	GVL.Pro4_.Signal_In.T_Ts_Result_Scanner( IN:= GVL.X[31], PT := T#0MS);
	GVL.Pro4_.Signal_In.T_Ts_Pass( IN:= GVL.X[21], PT := T#10MS);
	GVL.Pro4_.Signal_In.T_Ts_Fail( IN:= GVL.X[22], PT := T#10MS);
	GVL.Pro4_.Signal_In.T_Door_ss( IN:= GVL.X[23], PT := T#100MS);
	GVL.Pro4_.Signal_In.T_Ts_Press_Up( IN:= GVL.X[24], PT := T#10MS);
	GVL.Pro4_.Signal_In.T_Ts_Check_Gap( IN:= GVL.X[25], PT := T#500MS);
	// CHECK TS 
	T_RESET_TS(IN := GVL.Pro4_.Man.D_Ts = 2 OR GVL.Pro4_.Man.D_Ts = 3,  PT := T#5S, Q =>);
	T_OUT_RESET_TS( IN := (GVL.Y[20] AND NOT GVL.Pro4_.Signal_In.T_Ts_Fail.Q AND NOT  GVL.Pro4_.Signal_In.T_Ts_Pass.Q), PT := T#20S, Q =>);
	IF GVL.Y[20] AND GVL.Pro4_.Man.D_Ts = 0 AND NOT GVL.Pro4_.Signal_In.T_Ts_Fail.Q AND NOT GVL.Pro4_.Signal_In.T_Ts_Pass.Q  THEN
		GVL.Pro4_.Man.D_Ts := 1;
	END_IF;
	IF GVL.Pro4_.Man.D_Ts = 1 AND GVL.Pro4_.Signal_In.T_Ts_Pass.Q THEN
		GVL.Pro4_.Man.D_Ts := 2;
	ELSIF GVL.Pro4_.Man.D_Ts = 1 AND GVL.Pro4_.Signal_In.T_Ts_Fail.Q THEN
		GVL.Pro4_.Man.D_Ts := 3;
	END_IF
	IF T_RESET_TS.Q OR T_OUT_RESET_TS.Q THEN
		GVL.Pro4_.Man.TS_On_Off := 0;
		GVL.Pro4_.Man.D_Ts := 0 ;
		T_OUT_RESET_TS.IN := FALSE;
		T_RESET_TS.IN := FALSE;
	END_IF
	// check Víison
	GVL.Pro4_.Signal_In.T_Vs_detect( IN:= GVL.X[26], PT := T#100MS);
	GVL.Pro4_.Signal_In.T_Vs_Result_Scanner( IN:= GVL.X[30], PT := T#1MS);
	GVL.Pro4_.Signal_In.T_Vs_Pass( IN:= GVL.X[32] AND GVL.Pro4_.Signal_In.T_Vs_detect.Q, PT := T#1000MS);
	GVL.Pro4_.Signal_In.T_Vs_Fail( IN:= GVL.X[33] AND GVL.Pro4_.Signal_In.T_Vs_detect.Q, PT := T#1000MS);
	// CHECK VS 
	T_RESET_VS(IN := GVL.Pro4_.Man.D_Vs = 2 OR GVL.Pro4_.Man.D_Vs = 3,  PT := T#5S, Q =>);
	T_OUT_RESET_VS( IN := GVL.Y[21] AND NOT GVL.Pro4_.Signal_In.T_Vs_Fail.Q AND NOT  GVL.Pro4_.Signal_In.T_Vs_Pass.Q, PT := T#20S, Q =>);
	IF GVL.Y[21] AND GVL.Pro4_.Man.D_Vs = 0 AND NOT GVL.Pro4_.Signal_In.T_Vs_Fail.Q AND NOT GVL.Pro4_.Signal_In.T_Vs_Pass.Q  THEN
		GVL.Pro4_.Man.D_Vs := 1;
	END_IF;
	IF GVL.Pro4_.Man.D_Vs = 1 AND GVL.Pro4_.Signal_In.T_Ts_Pass.Q THEN
		GVL.Pro4_.Man.D_Vs := 2;
	ELSIF GVL.Pro4_.Man.D_Vs = 1 AND GVL.Pro4_.Signal_In.T_Ts_Fail.Q THEN
		GVL.Pro4_.Man.D_Vs := 3;
	END_IF
	IF T_RESET_VS.Q AND T_OUT_RESET_VS.Q THEN
		GVL.Pro4_.Man.Vs_On_Off := 0;
		GVL.Pro4_.Man.D_Vs := 0 ;
		T_OUT_RESET_VS.IN := FALSE;
		T_RESET_VS.IN := FALSE;
	END_IF
	// Conveyor
	GVL.Pro4_.Signal_In.T_Cv_In_1( IN:= NOT GVL.X[27], PT := T#1500MS);
	GVL.Pro4_.Signal_In.T_Cv_In_2( IN:= not GVL.X[28], PT := T#500MS);
	GVL.Pro4_.Signal_In.T_Cv_OK_out( IN:= GVL.X[29], PT := T#500MS);
	
	GVL.Pro4_.Signal_In.T_Cv_NG_out_1( IN:= NOT GVL.X[40], PT := T#10MS);
	GVL.Pro4_.Signal_In.T_Cv_NG_out_2( IN:= NOT GVL.X[41], PT := T#10MS);
	GVL.Pro4_.Signal_In.T_Cv_NG_out_full( IN:= NOT GVL.X[42], PT := T#10MS);

END_IF;


//


RETURN;
END_ACTION

ACTION ACT_Manual_MC:

END_ACTION

ACTION ACT_Out:
// Share all robot
// green
GVL.Y[2] := GVL.HMI_MAIN.yStart AND NOT GVL.HMI_MAIN.yStop AND NOT GVL.HMI_MAIN.yLamp_Yellow AND NOT POU_MOTION.HeavyAlarm ;
// red
GVL.Y[0] := GVL.HMI_MAIN.yStop AND NOT GVL.HMI_MAIN.yStart OR POU_MOTION.HeavyAlarm;
// yellow
GVL.Y[1] := GVL.HMI_MAIN.yLamp_Yellow OR POU_MOTION.LightAlarm;
// buzz
GVL.Y[3] := GVL.HMI_MAIN.yBuzz;

// Tool 1 A
GVL.Y[4] := GVL.RB_A_.Tool_1 OR GVL.Y[4];
// Tool 2 A
GVL.Y[5] := GVL.RB_A_.Tool_2;
// Tool 1 B			
GVL.Y[6] := GVL.RB_B_.Tool_1;
// Tool 2 B
GVL.Y[7] := GVL.RB_B_.Tool_2;

// Project 3
IF GVL.ProjectAndModel.Project_No_Current = 3 THEN
	
	// PRoject 4
	IF GVL.RB_A.Auto OR GVL.RB_B.Auto THEN
		GVL.Pro4_.Man.TS_On_Off := 0;
		GVL.Pro4_.Man.Vs_On_Off := 0;
		GVL.Pro4_.Man.Trigger_Barcode_Ts_On_Off := 0;
		GVL.Pro4_.Man.Trigger_Barcode_Ts_On_Off := 0;
		GVL.Pro4_.Man.Cv_NG_On_Off := 0;
		GVL.Pro4_.Man.Lighting_On_Off := 0;
		GVL.Pro4_.Man.centering_ts_On_Off := 0;
	END_IF
	
	IF GVL.RB_A.Manual OR GVL.RB_B.Manual THEN
		GVL.Pro4_.Auto.TS_On_Off := 0;
		GVL.Pro4_.Auto.Vs_On_Off := 0;
		GVL.Pro4_.Auto.Trigger_Barcode_Ts_On_Off := 0;
		GVL.Pro4_.Auto.Trigger_Barcode_Ts_On_Off := 0;
		GVL.Pro4_.Auto.Cv_NG_On_Off := 0;
		GVL.Pro4_.Auto.Lighting_On_Off := 0;
		GVL.Pro4_.Auto.centering_ts_On_Off := 0;
	END_IF
	
	// centering test sóng
	GVL.Y[10] :=  (GVL.RB_A.Auto AND GVL.RB_B.Auto AND GVL.Pro4_.Auto.centering_ts_On_Off )OR 
				( ( GVL.RB_A.Manual OR GVL.RB_B.Manual) AND GVL.Pro4_.Man.centering_ts_On_Off );
	
	// test sóng
	GVL.Y[20] :=  (GVL.RB_A.Auto AND GVL.RB_B.Auto AND GVL.Pro4_.Auto.TS_On_Off )OR 
				( ( GVL.RB_A.Manual OR GVL.RB_B.Manual) AND GVL.Pro4_.Man.TS_On_Off );
	// test vision			
	GVL.Y[21] :=  (GVL.RB_A.Auto AND GVL.RB_B.Auto AND GVL.Pro4_.Auto.Vs_On_Off )OR 
				( ( GVL.RB_A.Manual OR GVL.RB_B.Manual) AND GVL.Pro4_.Man.Vs_On_Off );
	// trigger Barcode	ts			
	GVL.Y[22] :=  (GVL.RB_A.Auto AND GVL.RB_B.Auto AND GVL.Pro4_.Auto.Trigger_Barcode_Ts_On_Off )OR 
				( ( GVL.RB_A.Manual OR GVL.RB_B.Manual) AND GVL.Pro4_.Man.Trigger_Barcode_Ts_On_Off );
	// trigger Barcode vs
	GVL.Y[23] :=  (GVL.RB_A.Auto AND GVL.RB_B.Auto AND GVL.Pro4_.Auto.Trigger_Barcode_Vs_On_Off )OR 
				( ( GVL.RB_A.Manual OR GVL.RB_B.Manual) AND GVL.Pro4_.Man.Trigger_Barcode_Vs_On_Off );
	// Conveyor NG
	GVL.Y[27] :=  (GVL.RB_A.Auto AND GVL.RB_B.Auto AND GVL.Pro4_.Auto.Cv_NG_On_Off )OR 
				( ( GVL.RB_A.Manual OR GVL.RB_B.Manual) AND GVL.Pro4_.Man.Cv_NG_On_Off );			
	// Lighting vision align
	GVL.Y[28] :=  (GVL.RB_A.Auto AND GVL.RB_B.Auto AND GVL.Pro4_.Auto.Lighting_On_Off )OR 
				( ( GVL.RB_A.Manual OR GVL.RB_B.Manual) AND GVL.Pro4_.Man.Lighting_On_Off );			
			
END_IF;
END_ACTION

ACTION ACT_SAVE_FILE:
// Duyet de kiem tra tin hieu luu va doc du lieu CAM
FOR i_cam := 0 TO 10 BY 1 DO
	GVL.RTrig_Save_Data_Cam[i_cam](CLK := GVL.Save_Data_Cam[i_cam]);
	GVL.RTrig_Load_Data_Cam[i_cam](CLK := GVL.Load_Data_Cam[i_cam]);
	// Luu du lieu CAM
	IF GVL.RTrig_Save_Data_Cam[i_cam].Q THEN
		filedata.Save(    
			pData := ADR(GVL.Data_Calib_RB),
			uiSize := SIZEOF(GVL.Data_Calib_RB),
			sFileName := CONCAT('Data_Cam_',INT_TO_STRING(i_cam)));
	END_IF
	// Doc lai du lieu CAM
	IF GVL.RTrig_Load_Data_Cam[i_cam].Q THEN
		filedata.Load(    
			pData := ADR(GVL.Data_Calib_RB),
			uiSize := SIZEOF(GVL.Data_Calib_RB),
			sFileName := CONCAT('Data_Cam_',INT_TO_STRING(i_cam)));
		GVL.Load_Data_Cam[i_cam] := FALSE;
	END_IF
END_FOR

// Save All Tool Config to File
r_Save_ToolConfig(CLK := GVL.g_stHMITool_Config_Save_All);
IF r_Save_ToolConfig.Q THEN
	
	filedata.Save(    
	pData := ADR(GVL.g_aToolConfigA),
    uiSize := SIZEOF(GVL.g_aToolConfigA),
    sFileName := 'Tool_Config_A.bin');	
	GVL.g_stHMITool_Config_Save_All := FALSE;
END_IF

// Read Tool Config From File
r_Read_ToolConfig(CLK := GVL.g_stHMITool_Config_Read_All);
IF r_Read_ToolConfig.Q OR Read_Config_First THEN
	
	filedata.Load(    
	pData := ADR(GVL.g_aToolConfigA),
    uiSize := SIZEOF(GVL.g_aToolConfigA),
    sFileName := 'Tool_Config_A.bin');	
	GVL.g_stHMITool_Config_Read_All := FALSE;
	GVL.g_stHMIToolEditorA.LoadCommand := TRUE; // cho doc du lieu tool hien tai
END_IF


// Save Conveyor Config
r_Save_ConveyorConfig(CLK:= GVL.g_stHMIConveyor_Config_Save);
IF r_Save_ConveyorConfig.Q THEN
	filedata.Save(    
	pData := ADR(GVL.g_aConveyorRuntime),
    uiSize := SIZEOF(GVL.g_aConveyorRuntime),
    sFileName := 'Conveyor_Config.bin');
	
END_IF

// Read Conveyor Config
r_Read_ConveyorConfig(CLK:= GVL.g_stHMIConveyor_Config_Read);
IF r_Read_ConveyorConfig.Q OR Read_Config_First THEN
	filedata.Load(    
	pData := ADR(GVL.g_aConveyorRuntime),
    uiSize := SIZEOF(GVL.g_aConveyorRuntime),
    sFileName := 'Conveyor_Config.bin');
	GVL.g_stHMIConveyor_Config_Read := FALSE;
END_IF

// Save Tracking Config
r_Save_TrackingConfig(CLK:= GVL.g_stHMITracking_Config_Save);
IF r_Save_TrackingConfig.Q THEN
	filedata.Save(    
	pData := ADR(GVL.g_stTrackingConfig_A),
    uiSize := SIZEOF(GVL.g_stTrackingConfig_A),
    sFileName := 'TrackingConfig_A.bin');
END_IF

// Read Tracking Config
r_Read_TrackingConfig(CLK:= GVL.g_stHMITracking_Config_Read);
IF r_Read_TrackingConfig.Q OR Read_Config_First THEN
	filedata.Load(    
	pData := ADR(GVL.g_stTrackingConfig_A),
    uiSize := SIZEOF(GVL.g_stTrackingConfig_A),
    sFileName := 'TrackingConfig_A.bin');
	GVL.g_stHMITracking_Config_Read := FALSE;
END_IF

// Save All Senssor Source Config to File
//r_Save_ToolConfig(CLK := GVL.g_stHMITool_Config_Save_All);
IF GVL.g_xHMISaveSensorSourceA_All THEN
	
	filedata.Save(    
	pData := ADR(GVL.g_aSensorSourceConfigA),
    uiSize := SIZEOF(GVL.g_aSensorSourceConfigA),
    sFileName := 'SensorSource_Config_A.bin');	
	GVL.g_xHMISaveSensorSourceA_All := FALSE;	
END_IF

// Read Tool Config From File
IF GVL.g_xHMILoadSensorSourceA_All OR Read_Config_First THEN
	
	filedata.Load(    
	pData := ADR(GVL.g_aSensorSourceConfigA),
    uiSize := SIZEOF(GVL.g_aSensorSourceConfigA),
    sFileName := 'SensorSource_Config_A.bin');	
	GVL.g_xHMILoadSensorSourceA_All := FALSE;
	GVL.g_xHMILoadSensorSourceA := TRUE; // cho doc du lieu senssor source hien tai
END_IF

// Save All Recipe Config to File
IF GVL.g_xHMISaveTrackingRecipeA_All THEN
	
	filedata.Save(    
	pData := ADR(GVL.g_aMultiTrackRecipeA),
    uiSize := SIZEOF(GVL.g_aMultiTrackRecipeA),
    sFileName := 'MultiTrackRecipe_Config_A.bin');	
	GVL.g_xHMISaveTrackingRecipeA_All := FALSE;	
END_IF

// Read Tool Config From File
IF GVL.g_xHMILoadTrackingRecipeA_All OR Read_Config_First THEN
	
	filedata.Load(    
	pData := ADR(GVL.g_aMultiTrackRecipeA),
    uiSize := SIZEOF(GVL.g_aMultiTrackRecipeA),
    sFileName := 'MultiTrackRecipe_Config_A.bin');	
	GVL.g_xHMILoadTrackingRecipeA_All := FALSE;
	GVL.g_xHMILoadTrackingRecipeA := TRUE; // cho doc du lieu senssor source hien tai
END_IF




//=============================================================================
// SAVE ALL VISION TRACKING SOURCE CONFIG
//=============================================================================
IF GVL.g_xHMISaveAllVisionSourceA THEN

    filedata.Save(
        pData := ADR(GVL.g_aVisionTrackingSourceConfigA),
        uiSize := SIZEOF(GVL.g_aVisionTrackingSourceConfigA),
        sFileName := 'VisionTrackingSource_Config_A.bin'
    );

    GVL.g_xHMISaveAllVisionSourceA := FALSE;

END_IF;


//=============================================================================
// LOAD ALL VISION TRACKING SOURCE CONFIG
//=============================================================================
IF GVL.g_xHMILoadAllVisionSourceA OR Read_Config_First THEN

    filedata.Load(
        pData := ADR(GVL.g_aVisionTrackingSourceConfigA),
        uiSize := SIZEOF(GVL.g_aVisionTrackingSourceConfigA),
        sFileName := 'VisionTrackingSource_Config_A.bin'
    );

    GVL.g_xHMILoadAllVisionSourceA := FALSE;

    // Sau khi đọc file, refresh Source đang hiển thị trên HMI.
    GVL.g_xHMILoadVisionSourceA := TRUE;

END_IF;


//=============================================================================
// ROBOT B - SAVE / LOAD TRACKING HMI CONFIG
// Parent: POU_Main -> ACT_SAVE_FILE
// Chèn block này TRƯỚC dòng: Read_Config_First := FALSE;
//=============================================================================

// Tool Config B.
IF GVL.g_xHMIToolConfigSaveAllB THEN
    filedata.Save(pData := ADR(GVL.g_aToolConfigB), uiSize := SIZEOF(GVL.g_aToolConfigB), sFileName := 'Tool_Config_B.bin');
    GVL.g_xHMIToolConfigSaveAllB := FALSE;
END_IF;

IF GVL.g_xHMIToolConfigReadAllB OR Read_Config_First THEN
    filedata.Load(pData := ADR(GVL.g_aToolConfigB), uiSize := SIZEOF(GVL.g_aToolConfigB), sFileName := 'Tool_Config_B.bin');
    GVL.g_xHMIToolConfigReadAllB := FALSE;
    GVL.g_stHMIToolEditorB.LoadCommand := TRUE;
END_IF;

// Tracking Config B.
IF GVL.g_xHMITrackingConfigSaveB THEN
    filedata.Save(pData := ADR(GVL.g_stTrackingConfig_B), uiSize := SIZEOF(GVL.g_stTrackingConfig_B), sFileName := 'TrackingConfig_B.bin');
    GVL.g_xHMITrackingConfigSaveB := FALSE;
END_IF;

IF GVL.g_xHMITrackingConfigReadB OR Read_Config_First THEN
    filedata.Load(pData := ADR(GVL.g_stTrackingConfig_B), uiSize := SIZEOF(GVL.g_stTrackingConfig_B), sFileName := 'TrackingConfig_B.bin');
    GVL.g_xHMITrackingConfigReadB := FALSE;
END_IF;

// Sensor Source B.
IF GVL.g_xHMISaveSensorSourceB_All THEN
    filedata.Save(pData := ADR(GVL.g_aSensorSourceConfigB), uiSize := SIZEOF(GVL.g_aSensorSourceConfigB), sFileName := 'SensorSource_Config_B.bin');
    GVL.g_xHMISaveSensorSourceB_All := FALSE;
END_IF;

IF GVL.g_xHMILoadSensorSourceB_All OR Read_Config_First THEN
    filedata.Load(pData := ADR(GVL.g_aSensorSourceConfigB), uiSize := SIZEOF(GVL.g_aSensorSourceConfigB), sFileName := 'SensorSource_Config_B.bin');
    GVL.g_xHMILoadSensorSourceB_All := FALSE;
    GVL.g_xHMILoadSensorSourceB := TRUE;
END_IF;

// Tracking Recipe B.
IF GVL.g_xHMISaveTrackingRecipeB_All THEN
    filedata.Save(pData := ADR(GVL.g_aMultiTrackRecipeB), uiSize := SIZEOF(GVL.g_aMultiTrackRecipeB), sFileName := 'MultiTrackRecipe_Config_B.bin');
    GVL.g_xHMISaveTrackingRecipeB_All := FALSE;
END_IF;

IF GVL.g_xHMILoadTrackingRecipeB_All OR Read_Config_First THEN
    filedata.Load(pData := ADR(GVL.g_aMultiTrackRecipeB), uiSize := SIZEOF(GVL.g_aMultiTrackRecipeB), sFileName := 'MultiTrackRecipe_Config_B.bin');
    GVL.g_xHMILoadTrackingRecipeB_All := FALSE;
    GVL.g_xHMILoadTrackingRecipeB := TRUE;
END_IF;

// Vision Tracking Source B.
IF GVL.g_xHMISaveAllVisionSourceB THEN
    filedata.Save(pData := ADR(GVL.g_aVisionTrackingSourceConfigB), uiSize := SIZEOF(GVL.g_aVisionTrackingSourceConfigB), sFileName := 'VisionTrackingSource_Config_B.bin');
    GVL.g_xHMISaveAllVisionSourceB := FALSE;
END_IF;

IF GVL.g_xHMILoadAllVisionSourceB OR Read_Config_First THEN
    filedata.Load(pData := ADR(GVL.g_aVisionTrackingSourceConfigB), uiSize := SIZEOF(GVL.g_aVisionTrackingSourceConfigB), sFileName := 'VisionTrackingSource_Config_B.bin');
    GVL.g_xHMILoadAllVisionSourceB := FALSE;
    GVL.g_xHMILoadVisionSourceB := TRUE;
END_IF;

// Tat bien doc du lieu khi khoi dong robot
Read_Config_First := FALSE;
END_ACTION

ACTION ACT_SelectProjectRun:
rSave_Model(CLK := GVL.Save_Model);
rCall_Model(CLK := GVL.Call_Model);
rReadModel_BF(CLK := Read_Model_BF);



IF rReadModel_BF.Q THEN
	filedata.Load(    
	pData := ADR(GVL.ProjectAndModel),
    uiSize := SIZEOF(GVL.ProjectAndModel),
    sFileName := 'ProjectAndModel_CR.bin');
	GVL.Project_No_Cur := GVL.ProjectAndModel.Project_No_Current;
	GVL.Model_No_Cur := GVL.ProjectAndModel.Model_No_Current;	
	
	S_Robot_Name_Full := CONCAT(S_Robot_Name,INT_TO_STRING(GVL.Project_No_Cur));
	S_Robot_Name_Full := CONCAT(S_Robot_Name_Full,'_Model_');
	S_Robot_Name_Full := CONCAT(S_Robot_Name_Full,INT_TO_STRING(GVL.Model_No_Cur));
	S_Robot_Name_Full := CONCAT(S_Robot_Name_Full,'.bin');
	
	filedata.Load(    
	pData := ADR(GVL.Robot_Programs[GVL.Project_No_Cur]),
    uiSize := SIZEOF(GVL.Robot_Programs[GVL.Project_No_Cur]),
    sFileName := S_Robot_Name_Full);
	
	
	GVL_1.DATA_RB_A := GVL.Robot_Programs[GVL.Project_No_Cur].Model[GVL.Model_No_Cur].DATA_RB_A;
	GVL_1.DATA_RB_B := GVL.Robot_Programs[GVL.Project_No_Cur].Model[GVL.Model_No_Cur].DATA_RB_B;
	GVL_1.Point_Name_A := GVL.Robot_Programs[GVL.Project_No_Cur].Point_Name_A;
	GVL_1.Point_Name_B := GVL.Robot_Programs[GVL.Project_No_Cur].Point_Name_B;
	GVL_1.Step_Cr_A := GVL.Robot_Programs[GVL.Project_No_Cur].Step_A;
	GVL_1.Step_Cr_B := GVL.Robot_Programs[GVL.Project_No_Cur].Step_B;
	GVL_1.Condition_Cr_A := GVL.Robot_Programs[GVL.Project_No_Cur].Condition_A;
	GVL_1.Condition_Cr_B := GVL.Robot_Programs[GVL.Project_No_Cur].Condition_B;
	GVL_1.StepCount_Cr_A := GVL.Robot_Programs[GVL.Project_No_Cur].StepCount_A;
	GVL_1.StepCount_Cr_B := GVL.Robot_Programs[GVL.Project_No_Cur].StepCount_B;
	GVL_1.CondCount_Cr_A := GVL.Robot_Programs[GVL.Project_No_Cur].CondCount_A;
	GVL_1.CondCount_Cr_B := GVL.Robot_Programs[GVL.Project_No_Cur].CondCount_B;
	GVL_1.Name_Program_Cr := GVL.Robot_Programs[GVL.Project_No_Cur].Name;
	
	GVL.A_LengthStep := GVL_1.StepCount_Cr_A;
	GVL.B_LengthStep := GVL_1.StepCount_Cr_B;
	
	Read_Model_BF := FALSE;
END_IF

// Tao bien Boolean xac nhan project dang chay
FOR i_1 := 0 TO 10 DO
	IF GVL.ProjectAndModel.Project_No_Current = i_1 THEN 
		IF GVL.ProjectAndModel.Direction_Robot_Current = 0 THEN
			GVL.Project_Cur[i_1] := TRUE;
		END_IF;
		IF GVL.ProjectAndModel.Direction_Robot_Current = 1 THEN
			GVL.Project_Cur_Rev[i_1] := TRUE;
		END_IF;
	ELSE
		IF GVL.ProjectAndModel.Direction_Robot_Current = 0 THEN
			GVL.Project_Cur[i_1] := FALSE;
		END_IF;
		IF GVL.ProjectAndModel.Direction_Robot_Current = 1 THEN
			GVL.Project_Cur_Rev[i_1] := FALSE;
		END_IF;
	END_IF
END_FOR

// Goi model
IF rCall_Model.Q THEN
	S_Robot_Name_Full := CONCAT(S_Robot_Name,INT_TO_STRING(GVL.Project_No_Cur));
	S_Robot_Name_Full := CONCAT(S_Robot_Name_Full,'_Model_');
	S_Robot_Name_Full := CONCAT(S_Robot_Name_Full,INT_TO_STRING(GVL.Model_No_Cur));
	S_Robot_Name_Full := CONCAT(S_Robot_Name_Full,'.bin');
	
	filedata.Load(    
	pData := ADR(GVL.Robot_Programs[GVL.Project_No_Cur]),
    uiSize := SIZEOF(GVL.Robot_Programs[GVL.Project_No_Cur]),
    sFileName := S_Robot_Name_Full);
	
	GVL_1.DATA_RB_A := GVL.Robot_Programs[GVL.Project_No_Cur].Model[GVL.Model_No_Cur].DATA_RB_A;
	GVL_1.DATA_RB_B := GVL.Robot_Programs[GVL.Project_No_Cur].Model[GVL.Model_No_Cur].DATA_RB_B;
	GVL_1.Point_Name_A := GVL.Robot_Programs[GVL.Project_No_Cur].Point_Name_A;
	GVL_1.Point_Name_B := GVL.Robot_Programs[GVL.Project_No_Cur].Point_Name_B;
	GVL_1.Step_Cr_A := GVL.Robot_Programs[GVL.Project_No_Cur].Step_A;
	GVL_1.Step_Cr_B := GVL.Robot_Programs[GVL.Project_No_Cur].Step_B;
	GVL_1.Condition_Cr_A := GVL.Robot_Programs[GVL.Project_No_Cur].Condition_A;
	GVL_1.Condition_Cr_B := GVL.Robot_Programs[GVL.Project_No_Cur].Condition_B;
	GVL_1.StepCount_Cr_A := GVL.Robot_Programs[GVL.Project_No_Cur].StepCount_A;
	GVL_1.StepCount_Cr_B := GVL.Robot_Programs[GVL.Project_No_Cur].StepCount_B;
	GVL_1.CondCount_Cr_A := GVL.Robot_Programs[GVL.Project_No_Cur].CondCount_A;
	GVL_1.CondCount_Cr_B := GVL.Robot_Programs[GVL.Project_No_Cur].CondCount_B;
	GVL_1.Name_Program_Cr := GVL.Robot_Programs[GVL.Project_No_Cur].Name;
	GVL.A_LengthStep := GVL_1.StepCount_Cr_A;
	GVL.B_LengthStep := GVL_1.StepCount_Cr_B;
	//GVL.Call_Model := FALSE;
END_IF

// Luu Model
IF rSave_Model.Q THEN
	S_Robot_Name_Full := CONCAT(S_Robot_Name,INT_TO_STRING(GVL.Project_No_Cur));
	S_Robot_Name_Full := CONCAT(S_Robot_Name_Full,'_Model_');
	S_Robot_Name_Full := CONCAT(S_Robot_Name_Full,INT_TO_STRING(GVL.Model_No_Cur));
	S_Robot_Name_Full := CONCAT(S_Robot_Name_Full,'.bin');
	
	GVL.ProjectAndModel.Project_No_Current := GVL.Project_No_Cur;
	GVL.ProjectAndModel.Model_No_Current := GVL.Model_No_Cur;
	
	GVL_1.StepCount_Cr_A := GVL.A_LengthStep;
	GVL_1.StepCount_Cr_B := GVL.B_LengthStep;
	
	GVL.Robot_Programs[GVL.Project_No_Cur].Model[GVL.Model_No_Cur].DATA_RB_A := GVL_1.DATA_RB_A;
	GVL.Robot_Programs[GVL.Project_No_Cur].Model[GVL.Model_No_Cur].DATA_RB_B := GVL_1.DATA_RB_B;

	GVL.Robot_Programs[GVL.Project_No_Cur].Point_Name_A := GVL_1.Point_Name_A;
	GVL.Robot_Programs[GVL.Project_No_Cur].Point_Name_B := GVL_1.Point_Name_B;
	GVL.Robot_Programs[GVL.Project_No_Cur].Step_A := GVL_1.Step_Cr_A;
	GVL.Robot_Programs[GVL.Project_No_Cur].Step_B := GVL_1.Step_Cr_B;
	GVL.Robot_Programs[GVL.Project_No_Cur].Condition_A := GVL_1.Condition_Cr_A;
	GVL.Robot_Programs[GVL.Project_No_Cur].Condition_B := GVL_1.Condition_Cr_B;
	GVL.Robot_Programs[GVL.Project_No_Cur].StepCount_A := GVL_1.StepCount_Cr_A;
	GVL.Robot_Programs[GVL.Project_No_Cur].StepCount_B := GVL_1.StepCount_Cr_B;
	GVL.Robot_Programs[GVL.Project_No_Cur].CondCount_A := GVL_1.CondCount_Cr_A;
	GVL.Robot_Programs[GVL.Project_No_Cur].CondCount_B := GVL_1.CondCount_Cr_B;
	GVL.Robot_Programs[GVL.Project_No_Cur].Name := GVL_1.Name_Program_Cr;

	filedata.Save(    
	pData := ADR(GVL.Robot_Programs[GVL.Project_No_Cur]),
    uiSize := SIZEOF(GVL.Robot_Programs[GVL.Project_No_Cur]),
    sFileName := S_Robot_Name_Full);
	
	filedata.Save(    
	pData := ADR(GVL.ProjectAndModel),
    uiSize := SIZEOF(GVL.ProjectAndModel),
    sFileName := 'ProjectAndModel_CR.bin');

END_IF
END_ACTION

ACTION ACT_StatusMode:
rTrig_Auto  (CLK := GVL.RB_A.Auto);
rTrig_Manual(CLK := GVL.RB_A.Manual);
rTrig_Lock  (CLK := GVL.RB_A.Lock);

IF rTrig_Auto.Q THEN
    GVL.RB_A.Manual := FALSE;
    GVL.RB_A.Lock   := FALSE;
END_IF;

IF rTrig_Manual.Q THEN
    GVL.RB_A.Auto := FALSE;
    GVL.RB_A.Lock := FALSE;
END_IF;

IF rTrig_Lock.Q THEN
    GVL.RB_A.Auto   := FALSE;
    GVL.RB_A.Manual := FALSE;
END_IF;

//////// 
rTrig_B_Auto  (CLK := GVL.RB_B.Auto);
rTrig_B_Manual(CLK := GVL.RB_B.Manual);
rTrig_B_Lock  (CLK := GVL.RB_B.Lock);

IF rTrig_B_Auto.Q THEN
    GVL.RB_B.Manual := FALSE;
    GVL.RB_B.Lock   := FALSE;
END_IF;

IF rTrig_B_Manual.Q THEN
    GVL.RB_B.Auto := FALSE;
    GVL.RB_B.Lock := FALSE;
END_IF;

IF rTrig_B_Lock.Q THEN
    GVL.RB_B.Auto   := FALSE;
    GVL.RB_B.Manual := FALSE;
END_IF;
END_ACTION

ACTION TimeTable:
// ================= RUN =================

GVL.TimeMachine.Run_H := TO_WORD(RunTime_s) / 3600;
GVL.TimeMachine.Run_M  := (TO_WORD(RunTime_s)  MOD 3600) / 60;
GVL.TimeMachine.Run_S   := TO_WORD(RunTime_s)  MOD 60;

// ================= STOP =================

GVL.TimeMachine.Stop_H  := TO_WORD(StopTime_s)/ 3600;
GVL.TimeMachine.Stop_M  := (TO_WORD(StopTime_s) MOD 3600) / 60;
GVL.TimeMachine.Stop_S  := TO_WORD(StopTime_s) MOD 60;

// ================= WAIT =================

GVL.TimeMachine.Wait_H  := TO_WORD(WaitTime_s) / 3600;
GVL.TimeMachine.Wait_M  := (TO_WORD(WaitTime_s) MOD 3600) / 60;
GVL.TimeMachine.Wait_S  := TO_WORD(WaitTime_s) MOD 60;

// ================= TOTAL =================
GVL.TimeMachine.Total_H  := TO_WORD(TotalTime_s)  / 3600;
GVL.TimeMachine.Total_M  := (TO_WORD(TotalTime_s)  MOD 3600) / 60;
GVL.TimeMachine.Total_S  := TO_WORD(TotalTime_s)  MOD 60;

// ================= TIMER 1S =================
T_1s(IN := TRUE, PT := T#1S);

IF T_1s.Q THEN
    Pulse_1s := TRUE;
    T_1s(IN := FALSE);
ELSE
    Pulse_1s := FALSE;
END_IF


// ================= ĐIỀU KIỆN CỘNG TGIAN =================
IF Pulse_1s AND NOT GVL.TimeMachine.CLEAR THEN
    // Tổng thời gian luôn tăng
    	TotalTime_s := TotalTime_s + 1;

    IF GVL.TimeMachine.Run THEN
        RunTime_s := RunTime_s + 1;
        
    ELSIF GVL.TimeMachine.Stop THEN
        StopTime_s := StopTime_s + 1;
        
    ELSIF GVL.TimeMachine.Wait THEN
        WaitTime_s := WaitTime_s + 1;        
    END_IF
ELSIF GVL.TimeMachine.CLEAR THEN
	TotalTime_s 	 := 0;
	RunTime_s		 := 0;
	StopTime_s		 := 0;
	WaitTime_s		 := 0;
END_IF
END_ACTION

END_PROGRAM

// Just_Motion_Control_x86_64_Linux_SM_WV/Application/FB_/FB_FileManager
FUNCTION_BLOCK PUBLIC FB_FileManager
VAR_INPUT
END_VAR
VAR_OUTPUT
END_VAR
VAR
	hFile    : SysFile.RTS_IEC_HANDLE;   //  file
    Result   : SysFile.RTS_IEC_RESULT;   // mã lỗi
    sPath    : STRING(200);      // đường dẫn file
END_VAR

METHOD Load : BOOL
VAR_INPUT
	pData : POINTER TO BYTE;
    uiSize : UDINT;
    sFileName : STRING;
END_VAR
VAR
	udiReadSize: UDINT;
END_VAR
// sPath := CONCAT('Data_Lock/', sFileName);
// 
// hFile := sysfile.SysFileOpen(
//     szFile := sPath,
//     am := ACCESS_MODE.AM_READ,
//     pResult := ADR(Result)
// );
// 
// IF hFile <> sysfile.RTS_INVALID_HANDLE THEN
// 
//     sysfile.SysFileRead(
//         hFile := hFile,
//         pbyBuffer := pData,
//         ulSize := uiSize,
//         pResult := ADR(Result)
//     );
// 
//     sysfile.SysFileClose(hFile);
// 
//     Load := TRUE;
// 
// ELSE
//     Load := FALSE;
// END_IF


//namnv0404
Load := FALSE;
Result := 0;
sPath := CONCAT('Data_Lock/', sFileName);

hFile := sysfile.SysFileOpen(
    szFile := sPath,
    am := sysfile.ACCESS_MODE.AM_READ,
    pResult := ADR(Result)
);

IF hFile <> sysfile.RTS_INVALID_HANDLE THEN

    udiReadSize := sysfile.SysFileRead(
        hFile := hFile,
        pbyBuffer := pData,
        ulSize := uiSize,
        pResult := ADR(Result)
    );

    sysfile.SysFileClose(hFile);

    IF (Result = 0) AND (udiReadSize = uiSize) THEN
        Load := TRUE;
    ELSE
        Load := FALSE;
    END_IF;

ELSE
    Load := FALSE;
END_IF;
END_METHOD

METHOD Save : BOOL
VAR_INPUT
	pData : POINTER TO BYTE;   // con trỏ dữ liệu
    uiSize : UDINT;            // kích thước
    sFileName : STRING;        // tên file
END_VAR
VAR
	udiWrittenSize: UDINT;
END_VAR
// // Ghép đường dẫn
// sPath := CONCAT('Data_Lock/', sFileName);
// 
// // 1️⃣ Mở file
// hFile := sysfile.SysFileOpen(
//     szFile := sPath,
//     am := sysfile.ACCESS_MODE.AM_WRITE_PLUS,
//     pResult := ADR(Result)
// );
// 
// 
// // 2️⃣ Nếu mở thành công thì ghi
// IF hFile <> sysfile.RTS_INVALID_HANDLE THEN
// 
//     sysfile.SysFileWrite(
//         hFile := hFile,
//         pbyBuffer := pData,
//         ulSize := uiSize,
//         pResult := ADR(Result)
//     );
// 
//     // 3️⃣ Đóng file
//     sysfile.SysFileClose(hFile);
// 
//     Save := TRUE;
// 
// ELSE
//     Save := FALSE;
// END_IF

//nmanv0404
Save := FALSE;
Result := 0;
sPath := CONCAT('Data_Lock/', sFileName);

hFile := sysfile.SysFileOpen(
    szFile := sPath,
    am := sysfile.ACCESS_MODE.AM_WRITE,
    pResult := ADR(Result)
);

IF hFile <> sysfile.RTS_INVALID_HANDLE THEN

    udiWrittenSize := sysfile.SysFileWrite(
        hFile := hFile,
        pbyBuffer := pData,
        ulSize := uiSize,
        pResult := ADR(Result)
    );

    sysfile.SysFileFlush(hFile);
    sysfile.SysFileClose(hFile);

    IF (Result = 0) AND (udiWrittenSize = uiSize) THEN
        Save := TRUE;
    ELSE
        Save := FALSE;
    END_IF;

ELSE
    Save := FALSE;
END_IF;
END_METHOD

END_FUNCTION_BLOCK

// Just_Motion_Control_x86_64_Linux_SM_WV/Application/PRG_ROBOT/POU_SAFETY_CHECK
PROGRAM POU_SAFETY_CHECK
VAR
	OVER_LIMIT_A, OVER_LIMIT_B, OVER_A_TO_B, OVER_B_TO_A, OVER_LIMIT_R : BOOL;
	
	LIMIT_A_X, LIMIT_A_Y, LIMIT_A_Z, LIMIT_A_R,
	LIMIT_B_X, LIMIT_B_Y, LIMIT_B_Z, LIMIT_B_R : BOOL;
END_VAR

ACT_RB_A();
ACT_RB_B();
// TRUC QUAY R
// IF GVL.M_R_.CUR_POS < TO_LREAL(GVL_1.DATA_M_R.LIMIT_BW) OR GVL.M_R_.CUR_POS > TO_LREAL(GVL_1.DATA_M_R.LIMIT_FW) THEN
// 	OVER_LIMIT_R := TRUE;
// 	ELSE
// 	OVER_LIMIT_R := FALSE;
// END_IF
// GVL.M_R_.SAFETY_CHECK := not OVER_LIMIT_R;

ACTION ACT_RB_A:
IF GVL.RB_A_.CUR_X >= TO_LREAL(GVL_1.DATA_RB_A.LIMIT_X_BW) AND 
	GVL.RB_A_.CUR_X <= TO_LREAL(GVL_1.DATA_RB_A.LIMIT_X_FW) THEN
	
	LIMIT_A_X := TRUE;
ELSE
	LIMIT_A_X := FALSE;
END_IF

IF GVL.RB_A_.CUR_Y >= TO_LREAL(GVL_1.DATA_RB_A.LIMIT_Y_BW) AND 
	GVL.RB_A_.CUR_Y <= TO_LREAL(GVL_1.DATA_RB_A.LIMIT_Y_FW) THEN
	
	LIMIT_A_Y := TRUE;
ELSE
	LIMIT_A_Y := FALSE;
END_IF
// IF GVL.RB_A_.CUR_Z < TO_LREAL(GVL_1.DATA_RB_A.LIMIT_Z_BW) OR GVL.RB_A_.CUR_Z > TO_LREAL(GVL_1.DATA_RB_A.LIMIT_Z_FW) THEN
// 	LIMIT_A_Z := TRUE;
// 	ELSE
// 	LIMIT_A_Z := FALSE;
// END_IF
// IF GVL.RB_A_.CUR_R < TO_LREAL(GVL_1.DATA_RB_A.LIMIT_R_BW) OR GVL.RB_A_.CUR_R > TO_LREAL(GVL_1.DATA_RB_A.LIMIT_R_FW) THEN
// 	LIMIT_A_R := TRUE;
// 	ELSE
// 	LIMIT_A_R := FALSE;
// END_IF
// OUT 1
IF LIMIT_A_X AND LIMIT_A_Y THEN
	OVER_LIMIT_A := TRUE;
ELSE
	OVER_LIMIT_A := FALSE;
END_IF
/// OUT 2
IF OVER_LIMIT_A  THEN
	GVL.RB_A_.SAFETY_CHECK := FALSE;
ELSE
	GVL.RB_A_.SAFETY_CHECK := TRUE;
END_IF
END_ACTION

ACTION ACT_RB_B:
IF GVL.RB_B_.CUR_X >= TO_LREAL(GVL_1.DATA_RB_B.LIMIT_X_BW) AND 
	GVL.RB_B_.CUR_X <= TO_LREAL(GVL_1.DATA_RB_B.LIMIT_X_FW) THEN
	
	LIMIT_B_X := TRUE;
ELSE
	LIMIT_B_X := FALSE;
END_IF

IF GVL.RB_B_.CUR_Y >= TO_LREAL(GVL_1.DATA_RB_B.LIMIT_Y_BW) AND 
	GVL.RB_B_.CUR_Y <= TO_LREAL(GVL_1.DATA_RB_B.LIMIT_Y_FW) THEN
	
	LIMIT_B_Y := TRUE;
ELSE
	LIMIT_B_Y := FALSE;
END_IF
// IF GVL.RB_B_.CUR_Z < TO_LREAL(GVL_1.DATA_RB_B.LIMIT_Z_BW) OR GVL.RB_B_.CUR_Z > TO_LREAL(GVL_1.DATA_RB_B.LIMIT_Z_FW) THEN
// 	LIMIT_B_Z := TRUE;
// 	ELSE
// 	LIMIT_B_Z := FALSE;
// END_IF
// IF GVL.RB_B_.CUR_R < TO_LREAL(GVL_1.DATA_RB_B.LIMIT_R_BW) OR GVL.RB_B_.CUR_R > TO_LREAL(GVL_1.DATA_RB_B.LIMIT_R_FW) THEN
// 	LIMIT_B_R := TRUE;
// 	ELSE
// 	LIMIT_B_R := FALSE;
// END_IF
// OUT 1
IF LIMIT_B_X AND LIMIT_B_Y THEN
	OVER_LIMIT_B := TRUE;
ELSE
	OVER_LIMIT_B := FALSE;
END_IF

/// OUT 2
IF OVER_LIMIT_B THEN
	GVL.RB_B_.SAFETY_CHECK := FALSE;
ELSE
	GVL.RB_B_.SAFETY_CHECK := TRUE;
END_IF
END_ACTION

END_PROGRAM

// Just_Motion_Control_x86_64_Linux_SM_WV/Application/FB_/FB_CONVERT_POS
FUNCTION_BLOCK FB_CONVERT_POS
VAR
END_VAR
VAR_INPUT
	POS_IN : SM3_Robotics.SMC_POS_REF;
END_VAR

VAR_OUTPUT
	X , Y , Z , A , B , C : REAL;
END_VAR

X := TO_REAL(POS_IN.c.X);
Y := TO_REAL(POS_IN.c.Y);
Z := TO_REAL(POS_IN.c.Z);
A := TO_REAL(POS_IN.c.A);
B := TO_REAL(POS_IN.c.B);
C := TO_REAL(POS_IN.c.C);

END_FUNCTION_BLOCK

// Just_Motion_Control_x86_64_Linux_SM_WV/Application/FB_/FB_RunMoveP_1
FUNCTION_BLOCK FB_RunMoveP_1
VAR_INPUT
    Start       : BOOL;
    
    Item        : ST_MotionQueueItem;
    PositionIn  : SMC_POS_REF;
    CoordSystem : SMC_COORD_SYSTEM;

    AcceptTimeoutTime : TIME := T#2S;
    MoveTimeoutTime   : TIME := T#10S;
    PosCheckDelayTime : TIME := T#100MS;
END_VAR

VAR_OUTPUT
    Accepted       : BOOL;
    Done           : BOOL;
    Busy           : BOOL;
    Active         : BOOL;
    Error          : BOOL;
    Timeout        : BOOL;
    Aborted        : BOOL;
    ErrorID        : SMC_ERROR;
    ErrorID_Custom : INT;
    State          : E_MoveState;
END_VAR
VAR_IN_OUT
	AxisGroup   : AXIS_GROUP_REF_SM3;
END_VAR
VAR
    fbMoveP : MC_MoveDirectAbsolute;

    tAcceptTimeout : TON;
    tMoveTimeout   : TON;
    tPosCheckDelay : TON;

    StartEdge    : BOOL;
    LastStart    : BOOL;
    ExecutePulse : BOOL;

    PosBuf : SMC_POS_REF;

    BufferMode : SM3_Robotics.MC_BUFFER_MODE;
    TransMode  : SM3_Robotics.MC_TRANSITION_MODE;
    TransParam : ARRAY[0..(SMC_RCNST.MAX_TRANS_PARAMS - 1)] OF LREAL := [0.0, 0.0];

    VelFacLocal    : LREAL;
    AccFacLocal    : LREAL;
    JerkFacLocal   : LREAL;
    TorqueFacLocal : LREAL;
END_VAR

VAR CONSTANT
    C_BM_Buffered     : SM3_Robotics.MC_BUFFER_MODE := 1;
    C_BM_BlendingNext : SM3_Robotics.MC_BUFFER_MODE := 4;

    C_TM_CornerDistance : SM3_Robotics.MC_TRANSITION_MODE := 2;
    C_TM_None           : SM3_Robotics.MC_TRANSITION_MODE := 0;
    C_TM_StartVelocity  : SM3_Robotics.MC_TRANSITION_MODE := 1;
END_VAR

//====================================================
// FB_RunMoveP
// Dùng cho MC_MoveDirectAbsolute
// MoveP KHÔNG có Velocity / Acc / Dec / Jerk
// Chỉ dùng VelFactor / AccFactor / JerkFactor / TorqueFactor
//====================================================

// Bắt cạnh lên Start
StartEdge := Start AND NOT LastStart;
LastStart := Start;

// Output dạng pulse
Accepted := FALSE;
Done := FALSE;
Timeout := FALSE;
Aborted := FALSE;

// Execute chỉ ON trong state MOVE_SEND
ExecutePulse := StartEdge;


// MoveP chỉ lấy Factor
VelFacLocal    := GVL_1.DATA_RB_A.Fac_Vel;
AccFacLocal    := GVL_1.DATA_RB_A.Fac_Acc;
JerkFacLocal   := GVL_1.DATA_RB_A.Fac_Jerk;
TorqueFacLocal := GVL_1.DATA_RB_A.Fac_Torque;

// Giá trị an toàn
IF VelFacLocal <= 0.0 THEN VelFacLocal := 0.1; END_IF;
IF AccFacLocal <= 0.0 THEN AccFacLocal := 0.1; END_IF;
IF JerkFacLocal <= 0.0 THEN JerkFacLocal := 0.1; END_IF;
IF TorqueFacLocal <= 0.0 THEN TorqueFacLocal := 0.1; END_IF;

// Mapping Blend


	// Không blend
	BufferMode := GVL.C_BM_Aborting;
	TransMode  := C_TM_None;
	TransParam[0] := 0.0;
	TransParam[1] := 0.0;




PosBuf := PositionIn;
//Gọi FB gốc
fbMoveP(
    AxisGroup := AxisGroup,
    Execute := Start,

    Position := PosBuf,
    CoordSystem := CoordSystem,

    BufferMode := BufferMode,
    TransitionMode := TransMode,
    TransitionParameter := TransParam,

    VelFactor := VelFacLocal,
    AccFactor := AccFacLocal,
    JerkFactor := JerkFacLocal,
    TorqueFactor := TorqueFacLocal
);

Busy := fbMoveP.Busy;
Active := fbMoveP.Active;

END_FUNCTION_BLOCK

// Just_Motion_Control_x86_64_Linux_SM_WV/Application/PRG_MACHINE/PRG_VisionTest
PROGRAM PRG_VisionTest
VAR
END_VAR
VAR
    diTestCapturePos : DINT;
END_VAR

//=============================================================================
// TEST - CAPTURE CONVEYOR POSITION
//-----------------------------------------------------------------------------
// Giả lập vị trí Encoder tại đúng thời điểm Camera chụp.
//=============================================================================
diTestCapturePos := F_VisionRealToRawDINT(
    Value := GVL.g_aConveyorRuntime[1].Status.PositionMM,
    Scale := GVL.g_aVisionConfig[1].PositionScale
);



//=============================================================================
// TEST VISION CAMERA 1
//-----------------------------------------------------------------------------
// Giả lập Vision trả 1 Tracking Object.
// PositionScale = 0.001.
//=============================================================================

//-------------------------------------------------------------------------
// STATUS + HEADER
//-------------------------------------------------------------------------
GVL.MODBUS[100] := WORD#16#0049;    // Bit0 Heartbeat + Bit3 ResultReady + Bit6 BlockReady.

GVL.MODBUS[101] := 1;               // JobID.
GVL.MODBUS[102] := 70;              // VIS_APP_CONVEYOR_PICK.
GVL.MODBUS[103] := 80;              // VIS_DATA_TRACK_OBJECT.

GVL.MODBUS[104] := 5;               // TriggerID LOW.
GVL.MODBUS[105] := 0;               // TriggerID HIGH.

GVL.MODBUS[106] := 20;              // VIS_RESULT_OK.
GVL.MODBUS[107] := 0;               // ErrorCode.

GVL.MODBUS[108] := 1;               // DataCount = 1.
GVL.MODBUS[109] := 1;               // BlockCount = 1.
GVL.MODBUS[110] := 1;               // BlockIndex = 1.
GVL.MODBUS[111] := 1;               // BlockDataCount = 1.

GVL.MODBUS[112] := 0;               // Checksum LOW.
GVL.MODBUS[113] := 0;               // Checksum HIGH.

GVL.MODBUS[114] := 0;               // CaptureConveyorPos LOW.
GVL.MODBUS[115] := 0;               // CaptureConveyorPos HIGH.

GVL.MODBUS[114] := F_VisionDINTLowWord(diTestCapturePos);
GVL.MODBUS[115] := F_VisionDINTHighWord(diTestCapturePos);

//-------------------------------------------------------------------------
// OBJECT 1
// X = 10 mm
// Y = -20 mm
// A = 90 deg
//-------------------------------------------------------------------------
GVL.MODBUS[132] := F_VisionDINTLowWord(20000);
GVL.MODBUS[133] := F_VisionDINTHighWord(20000);

GVL.MODBUS[134] := F_VisionDINTLowWord(-20000);
GVL.MODBUS[135] := F_VisionDINTHighWord(-20000);

GVL.MODBUS[136] := F_VisionDINTLowWord(90000);
GVL.MODBUS[137] := F_VisionDINTHighWord(90000);

GVL.MODBUS[138] := WORD#16#0003;     // Bit0 Valid + Bit1 AngleValid.
GVL.MODBUS[139] := 95;               // Score.
GVL.MODBUS[140] := 1;                // ProductClassID.

END_PROGRAM

// Just_Motion_Control_x86_64_Linux_SM_WV/Application/PRG_ROBOT/PRG_TestVisionAlign
PROGRAM PRG_TestVisionAlign
VAR
    xEnable : BOOL := TRUE;                     // Enable FB.
    xStart : BOOL := FALSE;                     // Phát cạnh lên để Start.
    xReset : BOOL := FALSE;                     // Reset test.

    fbVisionAlign : FB_VisionAlign;             // FB cần test.
END_VAR

//=============================================================================
// TEST FB_VisionAlign
//=============================================================================
fbVisionAlign(
    Enable := xEnable AND NOT xReset,
    Start := xStart,
    CameraID := 1,
    JobID := 1
);

// Reset bài test.
IF xReset THEN
    xStart := FALSE;
END_IF;

END_PROGRAM

// Just_Motion_Control_x86_64_Linux_SM_WV/Application/PRG_ROBOT/PRG_TestVisionTriggerResult
PROGRAM PRG_TestVisionTriggerResult
VAR
    //=========================================================
    // Lệnh test từ Watch/HMI
    //=========================================================
    xStartTest : BOOL;                      // Cạnh lên bắt đầu một chu trình Vision.
    xResetTest : BOOL;                      // Reset chu trình test.

    //=========================================================
    // State machine test
    //=========================================================
    iState : INT;                           // State hiện tại của chu trình test.

    //=========================================================
    // Điều khiển hai FB
    //=========================================================
    xStartTrigger : BOOL;                   // Start cho FB_TriggerVS.
    xStartWaitResult : BOOL;                // Start cho FB_VisionWaitResult.

    //=========================================================
    // FB Vision
    //=========================================================
    fbTriggerVS : FB_TriggerVS;             // Gửi Trigger và chờ TriggerDone.
    fbWaitResult : FB_VisionWaitResult;     // Chờ Result đúng TriggerID.

    //=========================================================
    // Kết quả test
    //=========================================================
    xTestDone : BOOL;                       // TRUE khi toàn bộ Trigger + Result hoàn thành.
    xTestError : BOOL;                      // TRUE nếu một trong hai FB lỗi.
    iTestErrorID : INT;                     // Mã lỗi tổng của test.
END_VAR

//=============================================================================
// PRG_TestVisionTriggerResult
// Test toàn bộ:
// Trigger -> TriggerDone -> ResultReady -> kiểm tra Result -> Done
//=============================================================================


//=============================================================================
// 1. CALL FB_TRIGGER
// Camera 1, Job 1, Application ALIGN chỉ dùng làm cấu hình test ban đầu.
//=============================================================================
fbTriggerVS(
    Enable := NOT xResetTest,
    Start := xStartTrigger,
    CameraID := 1,
    JobID := 1,
    Application := E_VisionApplication.VIS_APP_ALIGN,
    count_Vs_Align_max := 3,
    T_Delay_Trigger_time := 30,
    Trigger_Again := FALSE,
    Pass_Triger_VS_NG := FALSE,
    Mode_ByPass_VS := FALSE
);


//=============================================================================
// 2. CALL FB_WAIT_RESULT
// ExpectedTriggerID lấy trực tiếp từ Trigger vừa thực hiện.
//=============================================================================
fbWaitResult(
    Enable := TRUE,
    Start := xStartWaitResult,
    CameraID := 1,
    ExpectedTriggerID := fbTriggerVS.CurrentTriggerID,
    ExpectedJobID := 1,
    ExpectedApplication := E_VisionApplication.VIS_APP_ALIGN
);


//=============================================================================
// 3. RESET TEST
//=============================================================================
IF xResetTest THEN
    iState := 0;

    xStartTrigger := FALSE;
    xStartWaitResult := FALSE;

    xTestDone := FALSE;
    xTestError := FALSE;
    iTestErrorID := 0;

    xStartTest := FALSE;
END_IF;


//=============================================================================
// 4. TEST STATE MACHINE
//=============================================================================
CASE iState OF

    //-------------------------------------------------------------------------
    // STATE 0 - IDLE
    // Chờ lệnh bắt đầu test.
    //-------------------------------------------------------------------------
    0:
        xStartTrigger := FALSE;
        xStartWaitResult := FALSE;

        xTestDone := FALSE;
        xTestError := FALSE;
        iTestErrorID := 0;

        IF xStartTest THEN
            xStartTrigger := TRUE;
            iState := 10;
        END_IF;


    //-------------------------------------------------------------------------
    // STATE 10 - WAIT TRIGGER DONE
    // FB_TriggerVS gửi Trigger và chờ Vision xác nhận TriggerDone.
    //-------------------------------------------------------------------------
    10:
        IF fbTriggerVS.Error THEN
            xStartTrigger := FALSE;

            xTestError := TRUE;
            iTestErrorID := 100 + fbTriggerVS.ErrorID;

            iState := 900;

        ELSIF fbTriggerVS.DoneAll THEN
            // Trigger đã hoàn thành.
            // Giữ TriggerID hiện tại và chuyển sang chờ Result.
            xStartTrigger := FALSE;
            xStartWaitResult := TRUE;

            iState := 20;
        END_IF;


    //-------------------------------------------------------------------------
    // STATE 20 - WAIT VISION RESULT
    // Chờ Result đúng với TriggerID vừa gửi.
    //-------------------------------------------------------------------------
    20:
        IF fbWaitResult.Error THEN
            xStartWaitResult := FALSE;

            xTestError := TRUE;
            iTestErrorID := 200 + fbWaitResult.ErrorID;

            iState := 900;

        ELSIF fbWaitResult.Done THEN
            xStartWaitResult := FALSE;

            iState := 30;
        END_IF;


    //-------------------------------------------------------------------------
    // STATE 30 - TEST DONE
    // X/Y/A/Score hiện có thể xem trực tiếp từ fbWaitResult.
    //-------------------------------------------------------------------------
    30:
        xTestDone := TRUE;

        // Nhả Start để chuẩn bị cho chu trình tiếp theo.
        IF NOT xStartTest THEN
            iState := 0;
        END_IF;


    //-------------------------------------------------------------------------
    // STATE 900 - ERROR
    // Chờ nhả Start hoặc Reset.
    //-------------------------------------------------------------------------
    900:
        xStartTrigger := FALSE;
        xStartWaitResult := FALSE;

        IF NOT xStartTest THEN
            iState := 0;
        END_IF;

END_CASE;

END_PROGRAM

// Just_Motion_Control_x86_64_Linux_SM_WV/Application/PRG_ROBOT/PRG_VisionTrackingTest_A
PROGRAM PRG_VisionTrackingTest_A

VAR
    //=========================================================================
    // TEST CONTROL
    //=========================================================================
    xResetTest : BOOL;
    xStartTest : BOOL;

    rtResetTest : R_TRIG;
    rtStartTest : R_TRIG;

    uiTestState : UINT := 0;
    udiTestTriggerID : UDINT := 1;


    //=========================================================================
    // FRAME TEST
    //-------------------------------------------------------------------------
    // 1 = Frame chỉ có Object A.
    // 2 = Frame có Object A + Object B.
    //=========================================================================
    uiTestObjectCount : UINT := 1;


    //=========================================================================
    // OBJECT A
    //=========================================================================
    rTestObjectAXMM : REAL := 100.0;
    rTestObjectAYMM : REAL := -20.0;
    rTestObjectAADeg : REAL := 90.0;

    diTestObjectAXRaw : DINT;
    diTestObjectAYRaw : DINT;
    diTestObjectAARaw : DINT;


    //=========================================================================
    // OBJECT B
    //=========================================================================
    rTestObjectBXMM : REAL := 160.0;
    rTestObjectBYMM : REAL := -20.0;
    rTestObjectBADeg : REAL := 90.0;

    diTestObjectBXRaw : DINT;
    diTestObjectBYRaw : DINT;
    diTestObjectBARaw : DINT;


    //=========================================================================
    // CAPTURE
    //=========================================================================
    diTestCapturePos : DINT;
	rTestMoveMM : REAL := 0.0;
	uiTestFrame : UINT := 1;
	
	xAutoResponseTest : BOOL := FALSE;
	udiLastAutoCommandTriggerID : UDINT := 0;
	
	//=============================================================================
	// AUTO RESPONSE POSITION SIMULATION
	//=============================================================================
	xAutoBaseCaptureValid : BOOL := FALSE;
	lrAutoBaseCapturePosMM : LREAL := 0.0;
	lrAutoMoveMM : LREAL := 0.0;
	
	rAutoObjectABaseXMM : REAL := 100.0;
	rAutoObjectBBaseXMM : REAL := 160.0;

	uiAutoFrameCount : UINT := 0;
END_VAR

//=============================================================================
// PRG_VisionTrackingTest_A
//-----------------------------------------------------------------------------
// Test pipeline:
// Vision Modbus -> Driver -> Adapter -> ObjectSource -> Tracking Queue.
//
// uiTestObjectCount = 1:
//      Frame chỉ có Object A.
//
// uiTestObjectCount = 2:
//      Frame có Object A + Object B.
//
// Có thể thay đổi X/Y/A Online để mô phỏng Object di chuyển theo Conveyor.
//=============================================================================

rtResetTest(CLK := xResetTest);
rtStartTest(CLK := xStartTest);


//=============================================================================
// NHẬN LỆNH RESET
//=============================================================================
IF rtResetTest.Q THEN
    uiTestState := 10;
END_IF;


//=============================================================================
// NHẬN LỆNH START
//-----------------------------------------------------------------------------
// Không tự Clear Queue khi Start.
// Nhờ vậy có thể test:
// Frame 1 = A
// Frame 2 = A + B
// Frame 3 = A + B
//=============================================================================
IF rtStartTest.Q AND uiTestState = 0 THEN
    uiTestState := 100;
END_IF;


// rTestObjectAXMM := rTestObjectABaseXMM + rTestMoveMM;
// rTestObjectBXMM := rTestObjectBBaseXMM + rTestMoveMM;

//=============================================================================
// MANUAL TEST FRAME
//-----------------------------------------------------------------------------
// Chỉ dùng bộ Frame cố định khi test bằng tay.
// Auto Response sẽ tự tính tọa độ theo Conveyor.
//=============================================================================
IF NOT xAutoResponseTest THEN

    CASE uiTestFrame OF

        // Frame 1: chỉ A.
        1:
            uiTestObjectCount := 1;
            rTestObjectAXMM := 100.0;
            rTestObjectBXMM := 160.0;

        // Frame 2: A + B, dịch +50 mm.
        2:
            uiTestObjectCount := 2;
            rTestObjectAXMM := 150.0;
            rTestObjectBXMM := 210.0;

        // Frame 3: A + B, dịch thêm +50 mm.
        3:
            uiTestObjectCount := 2;
            rTestObjectAXMM := 200.0;
            rTestObjectBXMM := 260.0;

    END_CASE;

END_IF;

//=============================================================================
// AUTO RESPONSE TEST
//-----------------------------------------------------------------------------
// Khi Background Vision Trigger tạo Command mới, chương trình test tự động
// lấy TriggerID của Command đó để sinh Result giả lập.
// Không cần bấm xStartTest bằng tay.
//=============================================================================
IF xAutoResponseTest
AND uiTestState = 0
AND GVL.g_aVisionCommand[1].Execute
AND GVL.g_aVisionCommand[1].TriggerID <> 0
AND GVL.g_aVisionCommand[1].TriggerID <> udiLastAutoCommandTriggerID THEN

    // Lấy đúng TriggerID do Background Trigger vừa tạo.
    udiTestTriggerID := GVL.g_aVisionCommand[1].TriggerID;

    // Ghi nhớ Command đã xử lý để không giả lập lại cùng TriggerID.
    udiLastAutoCommandTriggerID := GVL.g_aVisionCommand[1].TriggerID;
	
	// Đếm số frame Auto đã phát.
    uiAutoFrameCount := uiAutoFrameCount + 1;

    // Đi vào State tạo Vision Result giả lập.
    uiTestState := 100;
END_IF;


//=============================================================================
// STATE MACHINE
//=============================================================================
CASE uiTestState OF


    //=========================================================================
    // 0 - IDLE
    //=========================================================================
    0:
        GVL.g_xResetTrackingObjectSourceA := FALSE;
        GVL.g_xClearTrackingQueueA := FALSE;


    //=========================================================================
    // 10 - RESET PIPELINE TEST
    //-------------------------------------------------------------------------
    // Reset ObjectSource / Adapter và Clear Queue.
    // Không reset TriggerID để tránh sử dụng lại Transaction cũ.
    //=========================================================================
    10:
		//---------------------------------------------------------------------
		// 0. RESET MỐC AUTO RESPONSE TEST
		//---------------------------------------------------------------------
		// Frame Auto đầu tiên sau Reset sẽ lấy lại vị trí Conveyor hiện tại
		// làm mốc mới.
		xAutoBaseCaptureValid := FALSE;
		lrAutoBaseCapturePosMM := 0.0;
		lrAutoMoveMM := 0.0;
		uiAutoFrameCount := 0;
	
        //---------------------------------------------------------------------
		// 1. Hạ ResultReady / BlockReady trước khi Reset.
		//---------------------------------------------------------------------
		GVL.MODBUS[100] := WORD#16#0001;     // Chỉ giữ Heartbeat.
	
		//---------------------------------------------------------------------
		// 2. Reset Adapter + Vision Object Source.
		//---------------------------------------------------------------------
		GVL.g_xResetTrackingObjectSourceA := TRUE;
	
		//---------------------------------------------------------------------
		// 3. Reset FB_VisionModbusDriver Camera 1.
		// Đây là phần trước đó còn thiếu.
		//---------------------------------------------------------------------
		GVL.g_aVisionCommand[1].Reset := TRUE;
	
		//---------------------------------------------------------------------
		// 4. Clear toàn bộ Tracking Queue.
		//---------------------------------------------------------------------
		GVL.g_xClearTrackingQueueA := TRUE;
	
		//---------------------------------------------------------------------
		// 5. Xóa Result runtime cũ.
		//---------------------------------------------------------------------
		GVL.g_aVisionResult[1].Header.Valid := FALSE;
		GVL.g_aVisionResult[1].TrackObjectResult.Valid := FALSE;
		GVL.g_aVisionResult[1].TrackObjectResult.ObjectCount := 0;
	
		GVL.g_aVisionTrackingMultiResultA[1].Valid := FALSE;
		GVL.g_aVisionTrackingMultiResultA[1].TriggerID := 0;

        uiTestState := 20;


    //=========================================================================
    // 20 - GIỮ RESET THÊM MỘT SCAN
    //=========================================================================
    20:
        // Giữ ResultReady thấp trong toàn bộ thời gian Reset.
		GVL.MODBUS[100] := WORD#16#0001;
	
		// Giữ Adapter/ObjectSource Reset.
		GVL.g_xResetTrackingObjectSourceA := TRUE;
	
		// Giữ Modbus Driver Reset.
		GVL.g_aVisionCommand[1].Reset := TRUE;

        uiTestState := 30;


    //=========================================================================
	// 30 - HOLD RESET THÊM MỘT SCAN
	//-------------------------------------------------------------------------
	30:
		GVL.MODBUS[100] := WORD#16#0001;
		GVL.g_xResetTrackingObjectSourceA := TRUE;
		GVL.g_aVisionCommand[1].Reset := TRUE;
	
		uiTestState := 35;
		
	//=========================================================================
	// 35 - RELEASE RESET
	//-------------------------------------------------------------------------
	35:
		// Nhả toàn bộ Reset.
		GVL.g_xResetTrackingObjectSourceA := FALSE;
		GVL.g_aVisionCommand[1].Reset := FALSE;
		GVL.g_xClearTrackingQueueA := FALSE;
	
		// Vẫn giữ ResultReady thấp thêm một scan sau khi nhả Reset.
		GVL.MODBUS[100] := WORD#16#0001;
	
		uiTestState := 40;


    //=========================================================================
    // 40 - VERIFY RESET
    //=========================================================================
    40:
        IF GVL.g_stTrackingQueue_A.ValidCount = 0 AND GVL.g_stTrackingQueue_A.NextObjectID = 0 THEN
            uiTestState := 0;
        END_IF;


    //=========================================================================
	// 100 - CHỐT CAPTURE POSITION + CHUẨN BỊ DATA
	//=========================================================================
	100:
	
		//=========================================================================
		// AUTO RESPONSE MODE - TEST 3C
		//-------------------------------------------------------------------------
		// Frame 1:
		//      chỉ có A.
		//
		// Frame 2 trở đi:
		//      có A + B.
		//
		// A và B cách nhau cố định 60 mm theo X.
		// Cả hai cùng dịch theo Conveyor.
		//=========================================================================
		IF xAutoResponseTest THEN
		
			//---------------------------------------------------------------------
			// Chốt mốc Conveyor ở frame Auto đầu tiên.
			//---------------------------------------------------------------------
			IF NOT xAutoBaseCaptureValid THEN
				lrAutoBaseCapturePosMM :=
					REAL_TO_LREAL(GVL.g_aVisionCommand[1].CaptureConveyorPos);
		
				xAutoBaseCaptureValid := TRUE;
			END_IF;
		
			//---------------------------------------------------------------------
			// Quãng đường Conveyor đã chạy từ frame đầu.
			//---------------------------------------------------------------------
			lrAutoMoveMM :=
				REAL_TO_LREAL(GVL.g_aVisionCommand[1].CaptureConveyorPos)
				- lrAutoBaseCapturePosMM;
		
			//---------------------------------------------------------------------
			// FRAME 1: chỉ có Object A.
			//---------------------------------------------------------------------
			IF uiAutoFrameCount = 1 THEN
				uiTestObjectCount := 1;
		
			//---------------------------------------------------------------------
			// FRAME 2 trở đi: Camera nhìn thấy A + B.
			//---------------------------------------------------------------------
			ELSE
				uiTestObjectCount := 2;
			END_IF;
		
			//---------------------------------------------------------------------
			// OBJECT A.
			//---------------------------------------------------------------------
			rTestObjectAXMM :=
				rAutoObjectABaseXMM
				+ LREAL_TO_REAL(lrAutoMoveMM);
		
			rTestObjectAYMM := -20.0;
			rTestObjectAADeg := 90.0;
		
			//---------------------------------------------------------------------
			// OBJECT B.
			// B luôn cách A +60 mm theo X.
			//---------------------------------------------------------------------
			rTestObjectBXMM := rTestObjectAXMM + 60.0;
			rTestObjectBYMM := -20.0;
			rTestObjectBADeg := 90.0;
		
			//---------------------------------------------------------------------
			// Capture Conveyor Position lấy đúng từ Background Trigger.
			//---------------------------------------------------------------------
			diTestCapturePos :=
				F_VisionRealToRawDINT(
					Value := GVL.g_aVisionCommand[1].CaptureConveyorPos,
					Scale := GVL.g_aVisionConfig[1].PositionScale
				);
	
		//---------------------------------------------------------------------
		// MANUAL MODE
		//---------------------------------------------------------------------
		ELSE
	
			diTestCapturePos :=
				F_VisionRealToRawDINT(
					Value := GVL.g_aConveyorRuntime[1].Status.PositionMM,
					Scale := GVL.g_aVisionConfig[1].PositionScale
				);
	
		END_IF;
	
	
		//---------------------------------------------------------------------
		// CONVERT OBJECT A
		//---------------------------------------------------------------------
		diTestObjectAXRaw := F_VisionRealToRawDINT(Value := rTestObjectAXMM, Scale := GVL.g_aVisionConfig[1].PositionScale);
		diTestObjectAYRaw := F_VisionRealToRawDINT(Value := rTestObjectAYMM, Scale := GVL.g_aVisionConfig[1].PositionScale);
		diTestObjectAARaw := F_VisionRealToRawDINT(Value := rTestObjectAADeg, Scale := GVL.g_aVisionConfig[1].AngleScale);
	
		//---------------------------------------------------------------------
		// CONVERT OBJECT B
		//---------------------------------------------------------------------
		diTestObjectBXRaw := F_VisionRealToRawDINT(Value := rTestObjectBXMM, Scale := GVL.g_aVisionConfig[1].PositionScale);
		diTestObjectBYRaw := F_VisionRealToRawDINT(Value := rTestObjectBYMM, Scale := GVL.g_aVisionConfig[1].PositionScale);
		diTestObjectBARaw := F_VisionRealToRawDINT(Value := rTestObjectBADeg, Scale := GVL.g_aVisionConfig[1].AngleScale);
	
		uiTestState := 110;


    //=========================================================================
    // 110 - TẠO FRAME VISION HOÀN CHỈNH
    //-------------------------------------------------------------------------
    // Ghi toàn bộ Header + Payload trước.
    // Chỉ bật ResultReady / BlockReady sau khi data đã hoàn chỉnh.
    //=========================================================================
    110:

        //---------------------------------------------------------------------
        // Tạm hạ Ready trong khi đang ghi Frame mới.
        //---------------------------------------------------------------------
        GVL.MODBUS[100] := WORD#16#0001;


        //---------------------------------------------------------------------
        // RESULT HEADER
        //---------------------------------------------------------------------
        GVL.MODBUS[101] := 1;                                           // JobID.
        GVL.MODBUS[102] := 70;                                          // VIS_APP_CONVEYOR_PICK.
        GVL.MODBUS[103] := 80;                                          // VIS_DATA_TRACK_OBJECT.

        GVL.MODBUS[104] := F_VisionUDINTLowWord(udiTestTriggerID);       // TriggerID LOW.
        GVL.MODBUS[105] := F_VisionUDINTHighWord(udiTestTriggerID);      // TriggerID HIGH.

        GVL.MODBUS[106] := 20;                                          // VIS_RESULT_OK.
        GVL.MODBUS[107] := 0;                                           // ErrorCode.

        GVL.MODBUS[108] := UINT_TO_WORD(uiTestObjectCount);              // Tổng Object trong Frame.
        GVL.MODBUS[109] := 1;                                           // BlockCount.
        GVL.MODBUS[110] := 1;                                           // BlockIndex.
        GVL.MODBUS[111] := UINT_TO_WORD(uiTestObjectCount);              // Object trong Block này.

        GVL.MODBUS[112] := 0;                                           // Checksum LOW.
        GVL.MODBUS[113] := 0;                                           // Checksum HIGH.


        //---------------------------------------------------------------------
        // CAPTURE CONVEYOR POSITION
        //---------------------------------------------------------------------
        GVL.MODBUS[114] := F_VisionDINTLowWord(diTestCapturePos);
        GVL.MODBUS[115] := F_VisionDINTHighWord(diTestCapturePos);


        //---------------------------------------------------------------------
        // OBJECT A - RECORD 1
        // Register 132..140 = 9 WORD.
        //---------------------------------------------------------------------
        GVL.MODBUS[132] := F_VisionDINTLowWord(diTestObjectAXRaw);
        GVL.MODBUS[133] := F_VisionDINTHighWord(diTestObjectAXRaw);

        GVL.MODBUS[134] := F_VisionDINTLowWord(diTestObjectAYRaw);
        GVL.MODBUS[135] := F_VisionDINTHighWord(diTestObjectAYRaw);

        GVL.MODBUS[136] := F_VisionDINTLowWord(diTestObjectAARaw);
        GVL.MODBUS[137] := F_VisionDINTHighWord(diTestObjectAARaw);

        GVL.MODBUS[138] := WORD#16#0003;                                 // Bit0 Valid + Bit1 AngleValid.
        GVL.MODBUS[139] := 95;                                          // Score.
        GVL.MODBUS[140] := 1;                                           // ProductClassID.


        //---------------------------------------------------------------------
        // OBJECT B - RECORD 2
        // Chỉ có hiệu lực khi uiTestObjectCount >= 2.
        // Register 141..149 = 9 WORD.
        //---------------------------------------------------------------------
        IF uiTestObjectCount >= 2 THEN
            GVL.MODBUS[141] := F_VisionDINTLowWord(diTestObjectBXRaw);
            GVL.MODBUS[142] := F_VisionDINTHighWord(diTestObjectBXRaw);

            GVL.MODBUS[143] := F_VisionDINTLowWord(diTestObjectBYRaw);
            GVL.MODBUS[144] := F_VisionDINTHighWord(diTestObjectBYRaw);

            GVL.MODBUS[145] := F_VisionDINTLowWord(diTestObjectBARaw);
            GVL.MODBUS[146] := F_VisionDINTHighWord(diTestObjectBARaw);

            GVL.MODBUS[147] := WORD#16#0003;                             // Bit0 Valid + Bit1 AngleValid.
            GVL.MODBUS[148] := 96;                                      // Score.
            GVL.MODBUS[149] := 1;                                       // ProductClassID.
        ELSE
            // Clear Record B để tránh nhìn nhầm dữ liệu cũ khi monitor.
            GVL.MODBUS[141] := 0;
            GVL.MODBUS[142] := 0;
            GVL.MODBUS[143] := 0;
            GVL.MODBUS[144] := 0;
            GVL.MODBUS[145] := 0;
            GVL.MODBUS[146] := 0;
            GVL.MODBUS[147] := 0;
            GVL.MODBUS[148] := 0;
            GVL.MODBUS[149] := 0;
        END_IF;


        //---------------------------------------------------------------------
        // DATA ĐÃ HOÀN CHỈNH -> BẬT RESULT READY + BLOCK READY.
        //---------------------------------------------------------------------
        GVL.MODBUS[100] := WORD#16#0049;

        uiTestState := 130;


    //=========================================================================
    // 130 - GIỮ FRAME CHO TỚI KHI ADAPTER NHẬN
    //-------------------------------------------------------------------------
    // POU_MODBUS có thể ghi đè vùng Vision -> Robot ở scan sau.
    // Vì vậy phải giữ lại toàn bộ Frame trong lúc chờ Adapter.
    //=========================================================================
    130:

        //---------------------------------------------------------------------
        // STATUS + HEADER
        //---------------------------------------------------------------------
        GVL.MODBUS[100] := WORD#16#0049;

        GVL.MODBUS[101] := 1;
        GVL.MODBUS[102] := 70;
        GVL.MODBUS[103] := 80;

        GVL.MODBUS[104] := F_VisionUDINTLowWord(udiTestTriggerID);
        GVL.MODBUS[105] := F_VisionUDINTHighWord(udiTestTriggerID);

        GVL.MODBUS[106] := 20;
        GVL.MODBUS[107] := 0;

        GVL.MODBUS[108] := UINT_TO_WORD(uiTestObjectCount);
        GVL.MODBUS[109] := 1;
        GVL.MODBUS[110] := 1;
        GVL.MODBUS[111] := UINT_TO_WORD(uiTestObjectCount);

        GVL.MODBUS[112] := 0;
        GVL.MODBUS[113] := 0;


        //---------------------------------------------------------------------
        // CAPTURE POSITION
        //---------------------------------------------------------------------
        GVL.MODBUS[114] := F_VisionDINTLowWord(diTestCapturePos);
        GVL.MODBUS[115] := F_VisionDINTHighWord(diTestCapturePos);


        //---------------------------------------------------------------------
        // OBJECT A
        //---------------------------------------------------------------------
        GVL.MODBUS[132] := F_VisionDINTLowWord(diTestObjectAXRaw);
        GVL.MODBUS[133] := F_VisionDINTHighWord(diTestObjectAXRaw);

        GVL.MODBUS[134] := F_VisionDINTLowWord(diTestObjectAYRaw);
        GVL.MODBUS[135] := F_VisionDINTHighWord(diTestObjectAYRaw);

        GVL.MODBUS[136] := F_VisionDINTLowWord(diTestObjectAARaw);
        GVL.MODBUS[137] := F_VisionDINTHighWord(diTestObjectAARaw);

        GVL.MODBUS[138] := WORD#16#0003;
        GVL.MODBUS[139] := 95;
        GVL.MODBUS[140] := 1;


        //---------------------------------------------------------------------
        // OBJECT B
        //---------------------------------------------------------------------
        IF uiTestObjectCount >= 2 THEN
            GVL.MODBUS[141] := F_VisionDINTLowWord(diTestObjectBXRaw);
            GVL.MODBUS[142] := F_VisionDINTHighWord(diTestObjectBXRaw);

            GVL.MODBUS[143] := F_VisionDINTLowWord(diTestObjectBYRaw);
            GVL.MODBUS[144] := F_VisionDINTHighWord(diTestObjectBYRaw);

            GVL.MODBUS[145] := F_VisionDINTLowWord(diTestObjectBARaw);
            GVL.MODBUS[146] := F_VisionDINTHighWord(diTestObjectBARaw);

            GVL.MODBUS[147] := WORD#16#0003;
            GVL.MODBUS[148] := 96;
            GVL.MODBUS[149] := 1;
        ELSE
            GVL.MODBUS[141] := 0;
            GVL.MODBUS[142] := 0;
            GVL.MODBUS[143] := 0;
            GVL.MODBUS[144] := 0;
            GVL.MODBUS[145] := 0;
            GVL.MODBUS[146] := 0;
            GVL.MODBUS[147] := 0;
            GVL.MODBUS[148] := 0;
            GVL.MODBUS[149] := 0;
        END_IF;


        //---------------------------------------------------------------------
        // CHỜ ADAPTER NHẬN ĐÚNG TRANSACTION.
        //---------------------------------------------------------------------
        IF GVL.g_aVisionTrackingMultiResultA[1].Valid AND GVL.g_aVisionTrackingMultiResultA[1].TriggerID = udiTestTriggerID THEN
            uiTestState := 140;
        END_IF;


    //=========================================================================
    // 140 - CHỜ OBJECT SOURCE XỬ LÝ FRAME
    //-------------------------------------------------------------------------
    // Không dùng NextObjectID > 0 để xác nhận nữa vì:
    // - Frame có thể chỉ chứa Duplicate.
    // - Duplicate không làm NextObjectID tăng.
    //
    // ResultAcceptedPulse xác nhận ObjectSource đã nhận transaction.
    //=========================================================================
    //=========================================================================
	// 140 - CHỜ OBJECT SOURCE XỬ LÝ ĐÚNG TRANSACTION
	//-------------------------------------------------------------------------
	// Không dùng ResultAcceptedPulse vì đây chỉ là Pulse 1 scan.
	// Dùng udiLastProcessedTriggerID để xác nhận Result hiện tại đã được
	// ObjectSource nhận và xử lý.
	//=========================================================================
	140:
		// Tiếp tục giữ ResultReady trong khi chờ ObjectSource.
		GVL.MODBUS[100] := WORD#16#0049;
	
		// ObjectSource đã nhận đúng TriggerID hiện tại.
		IF PRG_TrackingObjectSource_A.fbVisionSourceA[1].udiLastProcessedTriggerID = udiTestTriggerID THEN
			uiTestState := 150;
		END_IF;


    //=========================================================================
    // 150 - TEST DONE
    //-------------------------------------------------------------------------
    // TriggerID tăng cho Frame kế tiếp.
    // KHÔNG Clear Queue.
    //=========================================================================
    150:
        // Hạ ResultReady + BlockReady.
		// Chỉ giữ Heartbeat.
		GVL.MODBUS[100] := WORD#16#0001;
	
		uiTestState := 160;
	//=========================================================================
	// 160 - GIỮ RELEASE ÍT NHẤT MỘT SCAN
	//-------------------------------------------------------------------------
	160:
		GVL.MODBUS[100] := WORD#16#0001;
	
		uiTestState := 170;
	//=========================================================================
	// 170 - HOÀN THÀNH FRAME
	//-------------------------------------------------------------------------
	170:
// 		// Tăng TriggerID cho frame tiếp theo.
// 		udiTestTriggerID := udiTestTriggerID + 1;
// 		IF udiTestTriggerID = 0 THEN udiTestTriggerID := 1; END_IF;
		
		IF NOT xAutoResponseTest THEN
			// Manual Test:
			// chương trình test tự quản lý TriggerID.
			udiTestTriggerID := udiTestTriggerID + 1;
			IF udiTestTriggerID = 0 THEN udiTestTriggerID := 1; END_IF;
		END_IF;
	
		// Auto Response:
		// Không tăng TriggerID tại đây.
		// TriggerID tiếp theo phải lấy từ Background Vision Trigger.
	
		uiTestState := 0;	
		

END_CASE;

END_PROGRAM

// Just_Motion_Control_x86_64_Linux_SM_WV/Application/FB_/Vision/FB_VisionAlign_1
FUNCTION_BLOCK FB_VisionAlign_1
VAR_INPUT
    Enable : BOOL;                              // Cho phép FB hoạt động.
    Start : BOOL;                               // Cạnh lên bắt đầu một chu trình Vision Align.

    CameraID : UINT;                            // ID Camera sử dụng.
    JobID : UINT;                               // JobID của Vision Align.

    BypassOffsetCheck : BOOL;                   // TRUE = mode test, bỏ qua X/Y/A và ép Offset = 0.
    CheckScore : BOOL;                          // TRUE = kiểm tra Score, FALSE = bỏ qua Score khi test.
    MinScore : REAL;                            // Score nhỏ nhất được chấp nhận.

    MaxOffsetX : REAL;                          // Giới hạn Offset X tối đa cho phép.
    MaxOffsetY : REAL;                          // Giới hạn Offset Y tối đa cho phép.
    MaxOffsetA : REAL;                          // Giới hạn Offset A tối đa cho phép.

    ToleranceX : REAL;                          // Sai số X được coi là đã Align.
    ToleranceY : REAL;                          // Sai số Y được coi là đã Align.
    ToleranceA : REAL;                          // Sai số A được coi là đã Align.

    TriggerRetryMax : INT;                      // Số lần thử Trigger tối đa.
    TriggerDelayTime : INT;                     // Tham số Delay/Timeout dùng cho FB_TriggerVS.
END_VAR


VAR_OUTPUT
    Busy : BOOL;                                // FB đang thực hiện Align.
    Done : BOOL;                                // Chu trình Align hoàn thành.
    Error : BOOL;                               // Có lỗi.
    ErrorID : INT;                              // Mã lỗi của FB.

    CurrentTriggerID : UDINT;                   // TriggerID đang xử lý.

    ResultValid : BOOL;                         // Result Vision hợp lệ.
    ResultScore : REAL;                         // Score Vision trả về.
    ResultFeatureID : UINT;                     // FeatureID Vision trả về.
    ResultStatus : E_VisionResultStatus;        // Trạng thái Result Vision.

    RawOffsetX : REAL;                          // Offset X gốc Vision trả về.
    RawOffsetY : REAL;                          // Offset Y gốc Vision trả về.
    RawOffsetA : REAL;                          // Offset A gốc Vision trả về.

    RobotOffsetX : REAL;                        // Offset X dùng cho Robot.
    RobotOffsetY : REAL;                        // Offset Y dùng cho Robot.
    RobotOffsetA : REAL;                        // Offset A dùng cho Robot.

    InTolerance : BOOL;                         // TRUE = Offset đã nằm trong tolerance.
    NeedCorrectionMove : BOOL;                  // TRUE = cần Robot chạy correction.
    State : INT;                                // State hiện tại để monitor/debug.
END_VAR


VAR
    StartOld : BOOL;                            // Giá trị Start của scan trước.

    xStartTrigger : BOOL;                       // Start nội bộ cho FB_TriggerVS.
    xStartWaitResult : BOOL;                    // Start nội bộ cho FB_VisionWaitResult.

    fbTriggerVS : FB_TriggerVS;                 // FB phát Trigger Vision.
    fbWaitResult : FB_VisionWaitResult;         // FB chờ Vision Result.
END_VAR

//=============================================================================
// FB_VisionAlign
//-----------------------------------------------------------------------------
// Chức năng:
// 1. Trigger Camera.
// 2. Chờ Vision Result đúng TriggerID.
// 3. Kiểm tra Valid / Score.
// 4. Có thể Bypass kiểm tra X/Y/A khi test.
// 5. Kiểm tra MaxOffset.
// 6. Kiểm tra Tolerance.
// 7. Xuất NeedCorrectionMove nếu Robot cần chạy hiệu chỉnh.
//
// LƯU Ý:
// - Phiên bản này CHƯA tự chạy Motion.
// - RobotOffset hiện đang dùng trực tiếp RawOffset.
// - Sau khi test flow ổn sẽ bổ sung Camera -> Robot Transform.
//=============================================================================


//=============================================================================
// 1. FB TRIGGER VISION
//=============================================================================
fbTriggerVS(
    Enable := Enable,
    Start := xStartTrigger,
    CameraID := CameraID,
    JobID := JobID,
    Application := E_VisionApplication.VIS_APP_ALIGN,
    count_Vs_Align_max := TriggerRetryMax,
    T_Delay_Trigger_time := TriggerDelayTime,
    Trigger_Again := FALSE,
    Pass_Triger_VS_NG := FALSE,
    Mode_ByPass_VS := FALSE
);

CurrentTriggerID := fbTriggerVS.CurrentTriggerID;


//=============================================================================
// 2. FB WAIT VISION RESULT
//=============================================================================
fbWaitResult(
    Enable := Enable,
    Start := xStartWaitResult,
    CameraID := CameraID,
    ExpectedTriggerID := CurrentTriggerID,
    ExpectedJobID := JobID,
    ExpectedApplication := E_VisionApplication.VIS_APP_ALIGN
);


//=============================================================================
// 3. DISABLE
//=============================================================================
IF NOT Enable THEN
    State := 0;
    StartOld := FALSE;

    Busy := FALSE;
    Done := FALSE;
    Error := FALSE;
    ErrorID := 0;

    xStartTrigger := FALSE;
    xStartWaitResult := FALSE;

    CurrentTriggerID := 0;

    ResultValid := FALSE;
    ResultScore := 0.0;
    ResultFeatureID := 0;
    ResultStatus := E_VisionResultStatus.VIS_RESULT_NONE;

    RawOffsetX := 0.0;
    RawOffsetY := 0.0;
    RawOffsetA := 0.0;

    RobotOffsetX := 0.0;
    RobotOffsetY := 0.0;
    RobotOffsetA := 0.0;

    InTolerance := FALSE;
    NeedCorrectionMove := FALSE;

    RETURN;
END_IF;


//=============================================================================
// 4. STATE MACHINE
//=============================================================================
CASE State OF


    //=========================================================================
    // 0 - IDLE
    //-------------------------------------------------------------------------
    // Chờ cạnh lên của Start.
    //=========================================================================
    0:
        Busy := FALSE;
        Done := FALSE;
        Error := FALSE;
        ErrorID := 0;

        xStartTrigger := FALSE;
        xStartWaitResult := FALSE;

        ResultValid := FALSE;
        ResultScore := 0.0;
        ResultFeatureID := 0;
        ResultStatus := E_VisionResultStatus.VIS_RESULT_NONE;

        RawOffsetX := 0.0;
        RawOffsetY := 0.0;
        RawOffsetA := 0.0;

        RobotOffsetX := 0.0;
        RobotOffsetY := 0.0;
        RobotOffsetA := 0.0;

        InTolerance := FALSE;
        NeedCorrectionMove := FALSE;

        IF Start AND NOT StartOld THEN

            // Kiểm tra CameraID trước khi truy cập Array Vision.
            IF CameraID < 1 OR CameraID > GVL.C_MAX_VISION_CHANNELS THEN
                Error := TRUE;
                ErrorID := 1;                   // CameraID không hợp lệ.
                State := 900;

            ELSE
                Busy := TRUE;
                xStartTrigger := TRUE;
                State := 10;
            END_IF;

        END_IF;


    //=========================================================================
    // 10 - WAIT TRIGGER DONE
    //-------------------------------------------------------------------------
    // Chờ FB_TriggerVS hoàn tất Trigger handshake.
    //=========================================================================
    10:
        Busy := TRUE;

        IF fbTriggerVS.Error THEN
            xStartTrigger := FALSE;

            Error := TRUE;
            ErrorID := 100 + fbTriggerVS.ErrorID;
            State := 900;

        ELSIF fbTriggerVS.DoneAll THEN
            xStartTrigger := FALSE;

            // Bắt đầu chờ Result của đúng Trigger vừa phát.
            xStartWaitResult := TRUE;
            State := 20;
        END_IF;


    //=========================================================================
    // 20 - WAIT RESULT
    //-------------------------------------------------------------------------
    // Chờ Vision Result có cùng:
    // - CameraID
    // - JobID
    // - Application
    // - TriggerID
    //=========================================================================
    20:
        Busy := TRUE;

        IF fbWaitResult.Error THEN
            xStartWaitResult := FALSE;

            Error := TRUE;
            ErrorID := 200 + fbWaitResult.ErrorID;
            State := 900;

        ELSIF fbWaitResult.Done THEN
            xStartWaitResult := FALSE;

            //-----------------------------------------------------------------
            // Lưu thông tin chung của Result.
            //-----------------------------------------------------------------
            ResultValid := fbWaitResult.ResultValid;
            ResultScore := fbWaitResult.ResultScore;
            ResultFeatureID := fbWaitResult.ResultFeatureID;
            ResultStatus := fbWaitResult.ResultStatus;

            //-----------------------------------------------------------------
            // MODE TEST:
            // Không dùng X/Y/A Vision.
            // Ép toàn bộ Offset = 0 để test handshake nhanh.
            //-----------------------------------------------------------------
            IF BypassOffsetCheck THEN
                RawOffsetX := 0.0;
                RawOffsetY := 0.0;
                RawOffsetA := 0.0;

            //-----------------------------------------------------------------
            // MODE NORMAL:
            // Lấy dữ liệu X/Y/A thực tế từ Vision.
            //-----------------------------------------------------------------
            ELSE
                RawOffsetX := fbWaitResult.ResultX;
                RawOffsetY := fbWaitResult.ResultY;
                RawOffsetA := fbWaitResult.ResultA;
            END_IF;

            State := 30;
        END_IF;


    //=========================================================================
	// 30 - CHECK RESULT
	//-------------------------------------------------------------------------
	// BypassOffsetCheck = TRUE:
	// - Dùng để test handshake Vision.
	// - Không kiểm tra ResultValid.
	// - Không kiểm tra X/Y/A.
	// - Score chỉ kiểm tra khi CheckScore = TRUE.
	//
	// BypassOffsetCheck = FALSE:
	// - Chạy normal.
	// - Bắt buộc ResultValid = TRUE.
	// - Kiểm tra Score.
	// - Kiểm tra giới hạn X/Y/A.
	//=========================================================================
	30:
		//-------------------------------------------------------------------------
		// MODE TEST HANDSHAKE
		//-------------------------------------------------------------------------
		IF BypassOffsetCheck THEN
	
			// Có thể vẫn kiểm tra Score nếu người dùng yêu cầu.
			IF CheckScore AND ResultScore < MinScore THEN
				Error := TRUE;
				ErrorID := 302;                      // Score thấp hơn MinScore.
				State := 900;
			ELSE
				// Không kiểm tra Valid/X/Y/A trong mode test.
				RawOffsetX := 0.0;
				RawOffsetY := 0.0;
				RawOffsetA := 0.0;
				State := 40;
			END_IF;
	
		//-------------------------------------------------------------------------
		// MODE NORMAL
		//-------------------------------------------------------------------------
		ELSE
	
			IF NOT ResultValid THEN
				Error := TRUE;
				ErrorID := 301;                      // Vision Result không hợp lệ.
				State := 900;
	
			ELSIF CheckScore AND ResultScore < MinScore THEN
				Error := TRUE;
				ErrorID := 302;                      // Score thấp hơn MinScore.
				State := 900;
	
			ELSIF ABS(RawOffsetX) > MaxOffsetX THEN
				Error := TRUE;
				ErrorID := 303;                      // Offset X vượt giới hạn.
				State := 900;
	
			ELSIF ABS(RawOffsetY) > MaxOffsetY THEN
				Error := TRUE;
				ErrorID := 304;                      // Offset Y vượt giới hạn.
				State := 900;
	
			ELSIF ABS(RawOffsetA) > MaxOffsetA THEN
				Error := TRUE;
				ErrorID := 305;                      // Offset A vượt giới hạn.
				State := 900;
	
			ELSE
				State := 40;
			END_IF;
	
		END_IF;


    //=========================================================================
    // 40 - CAMERA OFFSET -> ROBOT OFFSET
    //-------------------------------------------------------------------------
    // Hiện tại chưa áp dụng Transform Camera -> Robot.
    //
    // Mode Test:
    // RobotOffset luôn = 0.
    //
    // Mode Normal:
    // Tạm copy RawOffset để test flow.
    // Sau này sẽ thay bằng phép Rotate Vector Camera -> Robot.
    //=========================================================================
    40:
        IF BypassOffsetCheck THEN
            RobotOffsetX := 0.0;
            RobotOffsetY := 0.0;
            RobotOffsetA := 0.0;

        ELSE
            RobotOffsetX := RawOffsetX;
            RobotOffsetY := RawOffsetY;
            RobotOffsetA := RawOffsetA;
        END_IF;

        State := 50;


    //=========================================================================
    // 50 - CHECK TOLERANCE
    //-------------------------------------------------------------------------
    // Xác định Robot đã nằm trong sai số cho phép hay chưa.
    //=========================================================================
    50:
        InTolerance :=
            ABS(RobotOffsetX) <= ToleranceX
            AND ABS(RobotOffsetY) <= ToleranceY
            AND ABS(RobotOffsetA) <= ToleranceA;

        //---------------------------------------------------------------------
        // Đã nằm trong Tolerance -> Align hoàn thành.
        //---------------------------------------------------------------------
        IF InTolerance THEN
            NeedCorrectionMove := FALSE;

            Busy := FALSE;
            Done := TRUE;

            State := 100;

        //---------------------------------------------------------------------
        // Chưa đạt -> báo Motion bên ngoài cần chạy Correction.
        //---------------------------------------------------------------------
        ELSE
            NeedCorrectionMove := TRUE;

            Busy := TRUE;
            State := 60;
        END_IF;


    //=========================================================================
    // 60 - WAIT CORRECTION MOVE
    //-------------------------------------------------------------------------
    // Phiên bản hiện tại CHƯA điều khiển Motion.
    //
    // State này chỉ dùng để xác nhận:
    // Vision Result hợp lệ nhưng Robot cần chạy correction.
    //
    // Phiên bản tiếp theo sẽ thêm:
    // - CorrectionMoveDone
    // - CorrectionMoveError
    // - Trigger Vision lại sau khi Robot Move xong.
    //=========================================================================
    60:
        Busy := TRUE;
        Done := FALSE;
        NeedCorrectionMove := TRUE;


    //=========================================================================
    // 100 - ALIGN DONE
    //-------------------------------------------------------------------------
    // Giữ Done cho tới khi Start được hạ.
    //=========================================================================
    100:
        Busy := FALSE;
        Done := TRUE;
        Error := FALSE;
        NeedCorrectionMove := FALSE;

        IF NOT Start THEN
            State := 0;
        END_IF;


    //=========================================================================
    // 900 - ERROR
    //-------------------------------------------------------------------------
    // Giữ lỗi cho tới khi Start được hạ.
    //=========================================================================
    900:
        Busy := FALSE;
        Done := FALSE;

        xStartTrigger := FALSE;
        xStartWaitResult := FALSE;

        NeedCorrectionMove := FALSE;

        IF NOT Start THEN
            Error := FALSE;
            ErrorID := 0;
            State := 0;
        END_IF;

END_CASE;


//=============================================================================
// 5. SAVE OLD SIGNAL
//=============================================================================
StartOld := Start;

END_FUNCTION_BLOCK

// Just_Motion_Control_x86_64_Linux_SM_WV/Application/FC_/Geometry/F_AngleBetweenPoints
FUNCTION F_AngleBetweenPoints : REAL
VAR_INPUT
    StartPos : ST_POS;    // Điểm bắt đầu.
    EndPos   : ST_POS;    // Điểm kết thúc.
END_VAR

VAR
    rDeltaX : REAL;       // Chênh lệch X.
    rDeltaY : REAL;       // Chênh lệch Y.
END_VAR

rDeltaX := EndPos.X - StartPos.X;
rDeltaY := EndPos.Y - StartPos.Y;

// ATAN2 trả kết quả theo radian, sau đó đổi sang độ.
F_AngleBetweenPoints :=
    F_RadToDeg(
        AngleRad := MyATAN2(rDeltaY, rDeltaX)
    );

END_FUNCTION

// Just_Motion_Control_x86_64_Linux_SM_WV/Application/FC_/Geometry/F_RadToDeg
FUNCTION F_RadToDeg : REAL
VAR_INPUT
    AngleRad : REAL;    // Góc đầu vào, đơn vị radian.
END_VAR

// Chuyển góc từ radian sang độ.
F_RadToDeg := AngleRad * GVL.C_RAD_TO_DEG;

END_FUNCTION

// Just_Motion_Control_x86_64_Linux_SM_WV/Application/FC_/Geometry/F_DegToRad
FUNCTION F_DegToRad  : REAL
VAR_INPUT
	AngleDeg : REAL;    // Góc đầu vào, đơn vị độ.
END_VAR
VAR
END_VAR

// Chuyển góc từ độ sang radian.
F_DegToRad := AngleDeg * GVL.C_DEG_TO_RAD;

END_FUNCTION

// Just_Motion_Control_x86_64_Linux_SM_WV/Application/FC_/Geometry/F_Distance2D
FUNCTION F_Distance2D : REAL
VAR_INPUT
    Pos1 : ST_POS;      // Điểm thứ nhất.
    Pos2 : ST_POS;      // Điểm thứ hai.
END_VAR

VAR
    rDeltaX : REAL;     // Chênh lệch tọa độ X.
    rDeltaY : REAL;     // Chênh lệch tọa độ Y.
END_VAR

// Tính độ lệch giữa hai điểm.
rDeltaX := Pos2.X - Pos1.X;
rDeltaY := Pos2.Y - Pos1.Y;

// Tính khoảng cách Euclid trong mặt phẳng XY.
F_Distance2D := SQRT(
    rDeltaX * rDeltaX
    + rDeltaY * rDeltaY
);

END_FUNCTION

// Just_Motion_Control_x86_64_Linux_SM_WV/Application/FC_/Geometry/F_Distance3D
FUNCTION F_Distance3D  : REAL
VAR_INPUT
    Pos1 : ST_POS;      // Điểm thứ nhất.
    Pos2 : ST_POS;      // Điểm thứ hai.
END_VAR

VAR
    rDeltaX : REAL;     // Chênh lệch tọa độ X.
    rDeltaY : REAL;     // Chênh lệch tọa độ Y.
    rDeltaZ : REAL;     // Chênh lệch tọa độ Z.
END_VAR

rDeltaX := Pos2.X - Pos1.X;
rDeltaY := Pos2.Y - Pos1.Y;
rDeltaZ := Pos2.Z - Pos1.Z;

// Tính khoảng cách trong không gian XYZ.
F_Distance3D := SQRT(
    rDeltaX * rDeltaX
    + rDeltaY * rDeltaY
    + rDeltaZ * rDeltaZ
);

END_FUNCTION

// Just_Motion_Control_x86_64_Linux_SM_WV/Application/FC_/Geometry/F_NormalizeAngleDeg
FUNCTION F_NormalizeAngleDeg  : REAL
VAR_INPUT
    AngleDeg : REAL;    // Góc cần chuẩn hóa, đơn vị độ.
END_VAR

VAR
    rResult : REAL;     // Giá trị góc sau chuẩn hóa.
END_VAR

// Sao chép góc đầu vào để xử lý.
rResult := AngleDeg;

// Đưa các góc lớn hơn 180 độ về vùng -180...180 độ.
WHILE rResult > 180.0 DO
    rResult := rResult - 360.0;
END_WHILE;

// Đưa các góc nhỏ hơn hoặc bằng -180 độ về vùng -180...180 độ.
WHILE rResult <= -180.0 DO
    rResult := rResult + 360.0;
END_WHILE;

F_NormalizeAngleDeg := rResult;

END_FUNCTION

// Just_Motion_Control_x86_64_Linux_SM_WV/Application/FC_/Geometry/F_NormalizeVector2D
FUNCTION F_NormalizeVector2D : ST_VECTOR_2D
VAR_INPUT
    Vector : ST_VECTOR_2D;    // Vector cần chuẩn hóa.
END_VAR

VAR
    rLength : REAL;           // Độ dài vector.
END_VAR

// Tính độ dài vector đầu vào.
rLength := F_VectorLength2D(Vector := Vector);

// Chỉ thực hiện phép chia khi độ dài đủ lớn.
IF rLength > GVL.C_REAL_EPSILON THEN
    F_NormalizeVector2D.X := Vector.X / rLength;
    F_NormalizeVector2D.Y := Vector.Y / rLength;
ELSE
    // Trả vector 0 nếu đầu vào không có hướng xác định.
    F_NormalizeVector2D.X := 0.0;
    F_NormalizeVector2D.Y := 0.0;
END_IF;

END_FUNCTION

// Just_Motion_Control_x86_64_Linux_SM_WV/Application/FC_/Geometry/F_VectorLength2D
FUNCTION F_VectorLength2D : REAL
VAR_INPUT
	Vector : ST_VECTOR_2D;    // Vector cần tính độ dài.
END_VAR
VAR
END_VAR

F_VectorLength2D := SQRT(
    Vector.X * Vector.X
    + Vector.Y * Vector.Y
);

END_FUNCTION

// Just_Motion_Control_x86_64_Linux_SM_WV/Application/FC_/Geometry/F_RotateAroundCenter2D
FUNCTION F_RotateAroundCenter2D : ST_POS
VAR_INPUT
    SourcePos : ST_POS;   // Điểm cần xoay.
    CenterPos : ST_POS;   // Tâm xoay.
    AngleDeg  : REAL;     // Góc xoay, đơn vị độ.
END_VAR

VAR
    stRelativePos : ST_POS;   // Tọa độ tương đối so với tâm.
    stRotatedPos  : ST_POS;   // Tọa độ sau khi xoay.
END_VAR

// Đưa điểm về hệ tọa độ có gốc tại tâm xoay.
stRelativePos.X := SourcePos.X - CenterPos.X;
stRelativePos.Y := SourcePos.Y - CenterPos.Y;
stRelativePos.Z := SourcePos.Z;
stRelativePos.A := SourcePos.A;

// Xoay điểm tương đối.
stRotatedPos := F_RotatePos2D(
    SourcePos := stRelativePos,
    AngleDeg := AngleDeg
);

// Chuyển điểm trở lại hệ tọa độ ban đầu.
F_RotateAroundCenter2D.X :=
    CenterPos.X + stRotatedPos.X;

F_RotateAroundCenter2D.Y :=
    CenterPos.Y + stRotatedPos.Y;

F_RotateAroundCenter2D.Z := stRotatedPos.Z;
F_RotateAroundCenter2D.A := stRotatedPos.A;

END_FUNCTION

// Just_Motion_Control_x86_64_Linux_SM_WV/Application/FC_/Geometry/F_RotatePos2D
FUNCTION F_RotatePos2D  : ST_POS
VAR_INPUT
    SourcePos : ST_POS;   // Điểm cần xoay.
    AngleDeg  : REAL;     // Góc xoay, đơn vị độ.
END_VAR

VAR
    rAngleRad : REAL;     // Góc xoay sau khi đổi sang radian.
    rCosAngle : REAL;     // Cosine góc xoay.
    rSinAngle : REAL;     // Sine góc xoay.
END_VAR

rAngleRad := F_DegToRad(AngleDeg := AngleDeg);
rCosAngle := COS(rAngleRad);
rSinAngle := SIN(rAngleRad);

// Xoay tọa độ X/Y quanh gốc.
F_RotatePos2D.X :=
    SourcePos.X * rCosAngle
    - SourcePos.Y * rSinAngle;

F_RotatePos2D.Y :=
    SourcePos.X * rSinAngle
    + SourcePos.Y * rCosAngle;

// Z không thay đổi trong phép xoay 2D.
F_RotatePos2D.Z := SourcePos.Z;

// Góc A của điểm được cộng thêm góc xoay.
F_RotatePos2D.A :=
    F_NormalizeAngleDeg(
        AngleDeg := SourcePos.A + AngleDeg
    );

END_FUNCTION

// Just_Motion_Control_x86_64_Linux_SM_WV/Application/FC_/Path/F_CalculateBlendRadius
FUNCTION F_CalculateBlendRadius : REAL
VAR_INPUT
    PreviousPos      : ST_POS;    // Điểm trước.
    CurrentPos       : ST_POS;    // Điểm hiện tại.
    NextPos          : ST_POS;    // Điểm sau.
    RequestedRadius  : REAL;      // Bán kính blend yêu cầu.
    MaxRatio         : REAL;      // Tỷ lệ tối đa so với đoạn ngắn nhất.
END_VAR

VAR
    rPreviousLength : REAL;    // Độ dài đoạn trước.
    rNextLength     : REAL;    // Độ dài đoạn sau.
    rMinLength      : REAL;    // Độ dài đoạn ngắn hơn.
    rRatio          : REAL;    // Tỷ lệ blend sau giới hạn.
END_VAR

rPreviousLength :=
    F_Distance3D(
        Pos1 := PreviousPos,
        Pos2 := CurrentPos
    );

rNextLength :=
    F_Distance3D(
        Pos1 := CurrentPos,
        Pos2 := NextPos
    );

// Chọn đoạn ngắn hơn để giới hạn bán kính blend.
IF rPreviousLength < rNextLength THEN
    rMinLength := rPreviousLength;
ELSE
    rMinLength := rNextLength;
END_IF;

// Giới hạn tỷ lệ hợp lệ từ 0 đến 0.5.
rRatio := LIMIT(0.0, MaxRatio, 0.5);

// Bán kính không được lớn hơn tỷ lệ cho phép của đoạn ngắn nhất.
F_CalculateBlendRadius :=
    MIN(RequestedRadius, rMinLength * rRatio);

END_FUNCTION

// Just_Motion_Control_x86_64_Linux_SM_WV/Application/FC_/Path/F_CalculatePathLength
FUNCTION F_CalculatePathLength : REAL
VAR_IN_OUT
    Path : ST_PATH_DATA;    // Path cần tính tổng chiều dài.
END_VAR

VAR
    uiIndex     : UINT;    // Chỉ số duyệt điểm.
    uiPointCount : UINT;   // Số điểm thực tế.
    rLength     : REAL;    // Tổng chiều dài path.
END_VAR

rLength := 0.0;
uiPointCount := Path.ProcessPointCount;

// Giới hạn số điểm theo kích thước array.
IF uiPointCount > GVL.C_MAX_PROCESS_PATH_POINTS THEN
    uiPointCount := GVL.C_MAX_PROCESS_PATH_POINTS;
END_IF;

// Path cần ít nhất hai điểm để có chiều dài.
IF uiPointCount >= 2 THEN
    FOR uiIndex := 2 TO uiPointCount DO
        rLength :=
            rLength
            + F_Distance3D(
                Pos1 := Path.ProcessPoints[uiIndex - 1].Pos,
                Pos2 := Path.ProcessPoints[uiIndex].Pos
            );
    END_FOR;
END_IF;

F_CalculatePathLength := rLength;

END_FUNCTION

// Just_Motion_Control_x86_64_Linux_SM_WV/Application/FC_/Path/F_InterpolatePosLinear
FUNCTION F_InterpolatePosLinear : ST_POS
VAR_INPUT
    StartPos : ST_POS;    // Điểm bắt đầu.
    EndPos   : ST_POS;    // Điểm kết thúc.
    Factor   : REAL;      // Hệ số nội suy 0...1.
END_VAR

VAR
    rFactor    : REAL;    // Hệ số sau giới hạn.
    rAngleDiff : REAL;    // Chênh lệch góc ngắn nhất.
END_VAR

rFactor := LIMIT(0.0, Factor, 1.0);

F_InterpolatePosLinear.X :=
    StartPos.X + (EndPos.X - StartPos.X) * rFactor;

F_InterpolatePosLinear.Y :=
    StartPos.Y + (EndPos.Y - StartPos.Y) * rFactor;

F_InterpolatePosLinear.Z :=
    StartPos.Z + (EndPos.Z - StartPos.Z) * rFactor;

// Nội suy góc theo hướng ngắn nhất qua biên ±180 độ.
rAngleDiff :=
    F_NormalizeAngleDeg(
        AngleDeg := EndPos.A - StartPos.A
    );

F_InterpolatePosLinear.A :=
    F_NormalizeAngleDeg(
        AngleDeg := StartPos.A + rAngleDiff * rFactor
    );

END_FUNCTION

// Just_Motion_Control_x86_64_Linux_SM_WV/Application/FC_/Path/F_IsDuplicatePathPoint
FUNCTION F_IsDuplicatePathPoint : BOOL
VAR_INPUT
    Point1           : ST_PATH_POINT;   // Điểm thứ nhất.
    Point2           : ST_PATH_POINT;   // Điểm thứ hai.
    MinDistance      : REAL;            // Khoảng cách nhỏ nhất, mm.
    MaxAngleDifference : REAL;          // Chênh lệch góc nhỏ nhất, độ.
END_VAR

VAR
    rDistance  : REAL;    // Khoảng cách hai điểm.
    rAngleDiff : REAL;    // Chênh lệch góc tuyệt đối.
END_VAR

rDistance :=
    F_PathPointDistance(
        Point1 := Point1,
        Point2 := Point2
    );

rAngleDiff :=
    ABS(
        F_NormalizeAngleDeg(
            AngleDeg := Point2.Pos.A - Point1.Pos.A
        )
    );

// Hai điểm được coi là trùng khi cả khoảng cách và góc đều rất nhỏ.
F_IsDuplicatePathPoint :=
    rDistance <= MinDistance
    AND rAngleDiff <= MaxAngleDifference;

END_FUNCTION

// Just_Motion_Control_x86_64_Linux_SM_WV/Application/FC_/Path/F_PathPointDistance
FUNCTION F_PathPointDistance  : REAL
VAR_INPUT
	Point1 : ST_PATH_POINT;    // Điểm path thứ nhất.
    Point2 : ST_PATH_POINT;    // Điểm path thứ hai.
END_VAR
VAR
END_VAR

F_PathPointDistance :=
    F_Distance3D(
        Pos1 := Point1.Pos,
        Pos2 := Point2.Pos
    );

END_FUNCTION

// Just_Motion_Control_x86_64_Linux_SM_WV/Application/FC_/Vision/F_CalcTraySlotTarget
FUNCTION F_CalcTraySlotTarget : ST_POS
VAR_INPUT
    MasterPos : ST_POS;
    RowCount : UINT;
    ColumnCount : UINT;
    RowPitchMM : REAL;
    ColumnPitchMM : REAL;
    FillByRow : BOOL;
    SlotIndex : UINT;
END_VAR

VAR
    uiRow : UINT;
    uiCol : UINT;
    rLocalX : REAL;
    rLocalY : REAL;
    rAngleRad : REAL;
    rCosA : REAL;
    rSinA : REAL;
END_VAR

// Mặc định trả lại Master; dữ liệu không hợp lệ thì không tính offset.
F_CalcTraySlotTarget := MasterPos;
IF SlotIndex = 0 OR RowCount = 0 OR ColumnCount = 0 THEN RETURN; END_IF;

// Tính Row/Column từ SlotIndex.
IF FillByRow THEN
    uiRow := ((SlotIndex - 1) / ColumnCount) + 1;
    uiCol := ((SlotIndex - 1) MOD ColumnCount) + 1;
ELSE
    uiCol := ((SlotIndex - 1) / RowCount) + 1;
    uiRow := ((SlotIndex - 1) MOD RowCount) + 1;
END_IF;

// Slot vượt kích thước Tray thì giữ nguyên Master để caller tự báo lỗi.
IF uiRow > RowCount OR uiCol > ColumnCount THEN RETURN; END_IF;

// Quy ước local Tray: +X theo Column, +Y theo Row.
rLocalX := UINT_TO_REAL(uiCol - 1) * ColumnPitchMM;
rLocalY := UINT_TO_REAL(uiRow - 1) * RowPitchMM;

// Rotate local offset theo góc A của Tray Master.
rAngleRad := MasterPos.A * GVL.C_DEG_TO_RAD;
rCosA := COS(rAngleRad);
rSinA := SIN(rAngleRad);

F_CalcTraySlotTarget.X := MasterPos.X + rLocalX * rCosA - rLocalY * rSinA;
F_CalcTraySlotTarget.Y := MasterPos.Y + rLocalX * rSinA + rLocalY * rCosA;
F_CalcTraySlotTarget.Z := MasterPos.Z;
F_CalcTraySlotTarget.A := MasterPos.A;

END_FUNCTION

// Just_Motion_Control_x86_64_Linux_SM_WV/Application/FC_/Vision/F_CheckAlignResult
FUNCTION F_CheckAlignResult  : BOOL
VAR_INPUT
	Result : ST_ALIGN_RESULT;    // Kết quả align cần kiểm tra.
    Config : ST_ALIGN_CONFIG;    // Giới hạn align.
END_VAR
VAR
END_VAR

F_CheckAlignResult :=
    Result.Valid
    AND Result.Score >= Config.MinScore
    AND ABS(Result.RobotOffset.X) <= Config.MaxOffsetX
    AND ABS(Result.RobotOffset.Y) <= Config.MaxOffsetY
    AND ABS(Result.RobotOffset.Z) <= Config.MaxOffsetZ
    AND ABS(Result.RobotOffset.A) <= Config.MaxOffsetA;

END_FUNCTION

// Just_Motion_Control_x86_64_Linux_SM_WV/Application/FC_/Vision/F_CheckPosRange
FUNCTION F_CheckPosRange : BOOL
VAR_INPUT
	Pos        : ST_POS;           // Tọa độ cần kiểm tra.
    RangeX     : ST_RANGE_REAL;    // Giới hạn X.
    RangeY     : ST_RANGE_REAL;    // Giới hạn Y.
    RangeZ     : ST_RANGE_REAL;    // Giới hạn Z.
    RangeA     : ST_RANGE_REAL;    // Giới hạn góc A.
END_VAR
VAR
END_VAR

F_CheckPosRange :=
    F_CheckRangeReal(
        Value := Pos.X,
        RangeConfig := RangeX
    )
    AND F_CheckRangeReal(
        Value := Pos.Y,
        RangeConfig := RangeY
    )
    AND F_CheckRangeReal(
        Value := Pos.Z,
        RangeConfig := RangeZ
    )
    AND F_CheckRangeReal(
        Value := Pos.A,
        RangeConfig := RangeA
    );

END_FUNCTION

// Just_Motion_Control_x86_64_Linux_SM_WV/Application/FC_/Vision/F_CheckRangeReal
FUNCTION F_CheckRangeReal : BOOL
VAR_INPUT
    Value       : REAL;             // Giá trị cần kiểm tra.
    RangeConfig : ST_RANGE_REAL;    // Cấu hình giới hạn.
END_VAR
VAR
END_VAR

IF NOT RangeConfig.Enable THEN
    // Bỏ qua kiểm tra khi giới hạn chưa được bật.
    F_CheckRangeReal := TRUE;
ELSE
    F_CheckRangeReal :=
        Value >= RangeConfig.MinValue
        AND Value <= RangeConfig.MaxValue;
END_IF;

END_FUNCTION

// Just_Motion_Control_x86_64_Linux_SM_WV/Application/FC_/Vision/F_CheckVisionHeader
FUNCTION F_CheckVisionHeader : BOOL
VAR_INPUT
	Header            : ST_VISION_RESULT_HEADER; // Header cần kiểm tra.
    ExpectedCameraID  : UINT;                    // Camera mong đợi.
    ExpectedJobID     : UINT;                    // Job mong đợi.
    ExpectedTriggerID : UDINT;                   // TriggerID mong đợi.
    MaxDataCount      : UINT;                    // Số phần tử tối đa.
END_VAR
VAR
END_VAR

// Header chỉ hợp lệ khi tất cả thông tin chính khớp yêu cầu.
F_CheckVisionHeader :=
    Header.Valid
    AND Header.CameraID = ExpectedCameraID
    AND Header.JobID = ExpectedJobID
    AND Header.TriggerID = ExpectedTriggerID
    AND Header.ErrorCode = 0
    AND Header.DataCount <= MaxDataCount;

END_FUNCTION

// Just_Motion_Control_x86_64_Linux_SM_WV/Application/FC_/Vision/F_CheckVisionScore
FUNCTION F_CheckVisionScore : BOOL
VAR_INPUT
	Score       : REAL;    // Score kết quả vision.
    MinScore    : REAL;    // Score nhỏ nhất được phép.
END_VAR
VAR
END_VAR

F_CheckVisionScore := Score >= MinScore;

END_FUNCTION

// Just_Motion_Control_x86_64_Linux_SM_WV/Application/FC_/Vision/F_CountInspectionFail
FUNCTION F_CountInspectionFail  : UINT
VAR_INPUT
    Result : ST_INSPECTION_RESULT;    // Kết quả inspection cần đếm.
END_VAR

VAR
    uiIndex     : UINT;    // Chỉ số duyệt các hạng mục.
    uiMaxCount  : UINT;    // Số item thực tế sau giới hạn.
    uiFailCount : UINT;    // Tổng số hạng mục không đạt.
END_VAR

uiFailCount := 0;

// Giới hạn số lượng để tránh vượt kích thước array.
uiMaxCount :=
    MIN(Result.ItemCount, GVL.C_MAX_INSPECTION_ITEMS);

FOR uiIndex := 1 TO uiMaxCount DO
    IF Result.Items[uiIndex].Valid
       AND NOT Result.Items[uiIndex].ResultOK THEN

        uiFailCount := uiFailCount + 1;
    END_IF;
END_FOR;

F_CountInspectionFail := uiFailCount;

END_FUNCTION
